SPLINE
SPL {X  -124.075, Y  +778.932, Z    +0.000, E1   -61.393, E3 +26417.862}
SPL {X  -150.653, Y  +735.257, Z    +0.000, E1   -50.160, E3 +26425.541}
SPL {X  -159.377, Y  +706.804, Z    +0.000, E1   -34.828, E3 +26427.184}
SPL {X  -162.134, Y  +688.425, Z    +0.000, E1   -19.100, E3 +26427.121}
SPL {X  -162.803, Y  +675.871, Z    +0.000, E1    -5.469, E3 +26427.305}
SPL {X  -162.820, Y  +671.500, Z    +0.000, E1    +0.000, E3 +26426.873}
SPL {X  -162.820, Y  +669.743, Z    +0.000, E1    +4.352, E3 +26426.669}
SPL {X  -162.820, Y  +665.917, Z    +0.000, E1   +15.272, E3 +26426.663}
SPL {X  -162.820, Y  +661.245, Z    +0.000, E1   +28.879, E3 +26426.504}
SPL {X  -162.820, Y  +654.015, Z    +0.000, E1   +45.814, E3 +26426.651}
SPL {X  -162.820, Y  +641.345, Z    +0.000, E1   +63.138, E3 +26426.698}
SPL {X  -162.820, Y  +620.039, Z    +0.000, E1   +75.979, E3 +26425.308}
SPL {X  -162.820, Y  +571.094, Z    +0.000, E1   +77.089, E3 +26440.487}
SPL {X  -157.487, Y  +339.169, Z    +0.000, E1   +76.425, E3 +26533.591}
SPL {X  -156.386, Y  +335.181, Z    +0.000, E1   +75.555, E3 +26545.652}
SPL {X  -152.710, Y  +324.020, Z    +0.000, E1   +75.365, E3 +26553.462}
SPL {X  -139.497, Y  +296.529, Z    +0.000, E1   +77.231, E3 +26547.034}
ENDSPLINE

SPLINE
SPL {X  -139.792, Y  +297.022, Z    +0.000, E1   +76.273, E3 +26555.729}
ENDSPLINE

SPLINE
SPL {X  -138.933, Y  +295.600, Z    +0.000, E1   +75.173, E3 +26566.212}
SPL {X  -137.186, Y  +292.805, Z    +0.000, E1   +73.993, E3 +26576.802}
SPL {X  -133.270, Y  +286.961, Z    +0.000, E1   +73.739, E3 +26581.515}
SPL {X  -130.283, Y  +282.844, Z    +0.000, E1   +73.297, E3 +26586.407}
SPL {X  -127.795, Y  +279.610, Z    +0.000, E1   +72.860, E3 +26590.537}
SPL {X  -124.650, Y  +275.749, Z    +0.000, E1   +72.674, E3 +26593.456}
SPL {X  -121.687, Y  +272.322, Z    +0.000, E1   +72.100, E3 +26597.765}
SPL {X  -113.980, Y  +264.229, Z    +0.000, E1   +74.120, E3 +26593.903}
SPL {X   -56.216, Y  +227.692, Z    +0.000, E1   +56.267, E3 +26770.627}
ENDSPLINE

SPLINE
SPL {X  -126.995, Y  +278.604, Z    +0.000, E1   +59.937, E3 +26942.868}
SPL {X  -150.196, Y  +317.640, Z    +0.000, E1   +49.956, E3 +26951.323}
SPL {X  -157.261, Y  +338.316, Z    +0.000, E1   +40.017, E3 +26953.018}
SPL {X  -160.924, Y  +355.726, Z    +0.000, E1   +27.715, E3 +26953.459}
SPL {X  -162.423, Y  +369.141, Z    +0.000, E1   +15.207, E3 +26953.894}
SPL {X  -162.811, Y  +378.755, Z    +0.000, E1    +4.616, E3 +26953.808}
SPL {X  -162.820, Y  +382.684, Z    +0.000, E1    -0.227, E3 +26953.363}
SPL {X  -162.820, Y  +387.227, Z    +0.000, E1   -12.320, E3 +26953.118}
SPL {X  -162.820, Y  +392.558, Z    +0.000, E1   -27.778, E3 +26953.154}
SPL {X  -162.820, Y  +400.474, Z    +0.000, E1   -46.251, E3 +26953.018}
SPL {X  -162.820, Y  +414.510, Z    +0.000, E1   -65.115, E3 +26952.461}
SPL {X  -162.820, Y  +465.064, Z    +0.000, E1   -76.269, E3 +26962.309}
SPL {X  -157.184, Y  +715.968, Z    +0.000, E1   -76.600, E3 +27058.266}
SPL {X  -156.461, Y  +718.560, Z    +0.000, E1   -75.553, E3 +27071.686}
SPL {X  -151.911, Y  +732.096, Z    +0.000, E1   -75.235, E3 +27082.240}
SPL {X  -146.569, Y  +744.407, Z    +0.000, E1   -74.677, E3 +27094.044}
SPL {X  -142.375, Y  +752.491, Z    +0.000, E1   -74.335, E3 +27101.072}
SPL {X  -139.539, Y  +757.399, Z    +0.000, E1   -73.892, E3 +27107.269}
SPL {X  -136.017, Y  +762.997, Z    +0.000, E1   -73.579, E3 +27112.452}
SPL {X  -133.089, Y  +767.296, Z    +0.000, E1   -73.251, E3 +27116.910}
SPL {X  -129.985, Y  +771.553, Z    +0.000, E1   -72.801, E3 +27121.904}
SPL {X  -126.581, Y  +775.909, Z    +0.000, E1   -72.426, E3 +27126.215}
SPL {X  -123.329, Y  +779.803, Z    +0.000, E1   -71.936, E3 +27130.597}
SPL {X  -119.291, Y  +784.315, Z    +0.000, E1   -72.148, E3 +27132.009}
SPL {X   -57.587, Y  +825.796, Z    +0.000, E1   -56.753, E3 +27285.771}
ENDSPLINE

SPLINE
SPL {X  -124.075, Y  +778.932, Z    +0.000, E1   -61.393, E3 +27479.400}
SPL {X  -150.653, Y  +735.257, Z    +0.000, E1   -50.160, E3 +27487.079}
SPL {X  -159.377, Y  +706.804, Z    +0.000, E1   -34.828, E3 +27488.723}
SPL {X  -162.134, Y  +688.425, Z    +0.000, E1   -19.100, E3 +27488.659}
SPL {X  -162.803, Y  +675.871, Z    +0.000, E1    -5.469, E3 +27488.843}
SPL {X  -162.820, Y  +671.500, Z    +0.000, E1    +0.000, E3 +27488.411}
SPL {X  -162.820, Y  +669.743, Z    +0.000, E1    +4.352, E3 +27488.207}
SPL {X  -162.820, Y  +665.917, Z    +0.000, E1   +15.272, E3 +27488.202}
SPL {X  -162.820, Y  +661.245, Z    +0.000, E1   +28.879, E3 +27488.043}
SPL {X  -162.820, Y  +654.015, Z    +0.000, E1   +45.814, E3 +27488.190}
SPL {X  -162.820, Y  +641.345, Z    +0.000, E1   +63.138, E3 +27488.237}
SPL {X  -162.820, Y  +620.039, Z    +0.000, E1   +75.979, E3 +27486.847}
SPL {X  -162.820, Y  +571.094, Z    +0.000, E1   +77.089, E3 +27502.025}
SPL {X  -157.487, Y  +339.169, Z    +0.000, E1   +76.425, E3 +27595.129}
SPL {X  -156.386, Y  +335.181, Z    +0.000, E1   +75.555, E3 +27607.190}
SPL {X  -152.710, Y  +324.020, Z    +0.000, E1   +75.365, E3 +27615.000}
SPL {X  -139.497, Y  +296.529, Z    +0.000, E1   +77.231, E3 +27608.572}
ENDSPLINE

SPLINE
SPL {X  -139.792, Y  +297.022, Z    +0.000, E1   +76.273, E3 +27617.267}
ENDSPLINE

SPLINE
SPL {X  -138.933, Y  +295.600, Z    +0.000, E1   +75.173, E3 +27627.750}
SPL {X  -137.186, Y  +292.805, Z    +0.000, E1   +73.993, E3 +27638.340}
SPL {X  -133.270, Y  +286.961, Z    +0.000, E1   +73.739, E3 +27643.054}
SPL {X  -130.283, Y  +282.844, Z    +0.000, E1   +73.297, E3 +27647.946}
SPL {X  -127.795, Y  +279.610, Z    +0.000, E1   +72.860, E3 +27652.076}
SPL {X  -124.650, Y  +275.749, Z    +0.000, E1   +72.674, E3 +27654.994}
SPL {X  -121.687, Y  +272.322, Z    +0.000, E1   +72.100, E3 +27659.304}
SPL {X  -113.980, Y  +264.229, Z    +0.000, E1   +74.120, E3 +27655.442}
SPL {X   -56.216, Y  +227.692, Z    +0.000, E1   +56.267, E3 +27832.166}
ENDSPLINE

SPLINE
SPL {X  -126.995, Y  +278.604, Z    +0.000, E1   +59.937, E3 +28004.406}
SPL {X  -150.196, Y  +317.640, Z    +0.000, E1   +49.956, E3 +28012.861}
SPL {X  -157.261, Y  +338.316, Z    +0.000, E1   +40.017, E3 +28014.556}
SPL {X  -160.924, Y  +355.726, Z    +0.000, E1   +27.715, E3 +28014.997}
SPL {X  -162.423, Y  +369.141, Z    +0.000, E1   +15.207, E3 +28015.432}
SPL {X  -162.811, Y  +378.755, Z    +0.000, E1    +4.616, E3 +28015.347}
SPL {X  -162.820, Y  +382.684, Z    +0.000, E1    -0.227, E3 +28014.902}
SPL {X  -162.820, Y  +387.227, Z    +0.000, E1   -12.320, E3 +28014.656}
SPL {X  -162.820, Y  +392.558, Z    +0.000, E1   -27.778, E3 +28014.692}
SPL {X  -162.820, Y  +400.474, Z    +0.000, E1   -46.251, E3 +28014.556}
SPL {X  -162.820, Y  +414.510, Z    +0.000, E1   -65.115, E3 +28013.999}
SPL {X  -162.820, Y  +465.064, Z    +0.000, E1   -76.269, E3 +28023.847}
SPL {X  -157.184, Y  +715.968, Z    +0.000, E1   -76.600, E3 +28119.805}
SPL {X  -156.461, Y  +718.560, Z    +0.000, E1   -75.553, E3 +28133.225}
SPL {X  -151.911, Y  +732.096, Z    +0.000, E1   -75.235, E3 +28143.779}
SPL {X  -146.569, Y  +744.407, Z    +0.000, E1   -74.677, E3 +28155.583}
SPL {X  -142.375, Y  +752.491, Z    +0.000, E1   -74.335, E3 +28162.610}
SPL {X  -139.539, Y  +757.399, Z    +0.000, E1   -73.892, E3 +28168.808}
SPL {X  -136.017, Y  +762.997, Z    +0.000, E1   -73.579, E3 +28173.990}
SPL {X  -133.089, Y  +767.296, Z    +0.000, E1   -73.251, E3 +28178.448}
SPL {X  -129.985, Y  +771.553, Z    +0.000, E1   -72.801, E3 +28183.442}
SPL {X  -126.581, Y  +775.909, Z    +0.000, E1   -72.426, E3 +28187.753}
SPL {X  -123.329, Y  +779.803, Z    +0.000, E1   -71.936, E3 +28192.135}
SPL {X  -119.291, Y  +784.315, Z    +0.000, E1   -72.148, E3 +28193.547}
SPL {X   -57.587, Y  +825.796, Z    +0.000, E1   -56.753, E3 +28347.309}
ENDSPLINE

SPLINE
SPL {X  -124.075, Y  +778.932, Z    +0.000, E1   -61.393, E3 +28540.938}
SPL {X  -150.653, Y  +735.257, Z    +0.000, E1   -50.160, E3 +28548.618}
SPL {X  -159.377, Y  +706.804, Z    +0.000, E1   -34.828, E3 +28550.261}
SPL {X  -162.134, Y  +688.425, Z    +0.000, E1   -19.100, E3 +28550.198}
SPL {X  -162.803, Y  +675.871, Z    +0.000, E1    -5.469, E3 +28550.382}
SPL {X  -162.820, Y  +671.500, Z    +0.000, E1    +0.000, E3 +28549.950}
SPL {X  -162.820, Y  +669.743, Z    +0.000, E1    +4.352, E3 +28549.746}
SPL {X  -162.820, Y  +665.917, Z    +0.000, E1   +15.272, E3 +28549.740}
SPL {X  -162.820, Y  +661.245, Z    +0.000, E1   +28.879, E3 +28549.581}
SPL {X  -162.820, Y  +654.015, Z    +0.000, E1   +45.814, E3 +28549.728}
SPL {X  -162.820, Y  +641.345, Z    +0.000, E1   +63.138, E3 +28549.775}
SPL {X  -162.820, Y  +620.039, Z    +0.000, E1   +75.979, E3 +28548.385}
SPL {X  -162.820, Y  +571.094, Z    +0.000, E1   +77.089, E3 +28563.564}
SPL {X  -157.487, Y  +339.169, Z    +0.000, E1   +76.425, E3 +28656.668}
SPL {X  -156.386, Y  +335.181, Z    +0.000, E1   +75.555, E3 +28668.729}
SPL {X  -152.710, Y  +324.020, Z    +0.000, E1   +75.365, E3 +28676.539}
SPL {X  -139.497, Y  +296.529, Z    +0.000, E1   +77.231, E3 +28670.111}
ENDSPLINE

SPLINE
SPL {X  -139.792, Y  +297.022, Z    +0.000, E1   +76.273, E3 +28678.806}
ENDSPLINE

SPLINE
SPL {X  -138.933, Y  +295.600, Z    +0.000, E1   +75.173, E3 +28689.289}
SPL {X  -137.186, Y  +292.805, Z    +0.000, E1   +73.993, E3 +28699.879}
SPL {X  -133.270, Y  +286.961, Z    +0.000, E1   +73.739, E3 +28704.592}
SPL {X  -130.283, Y  +282.844, Z    +0.000, E1   +73.297, E3 +28709.484}
SPL {X  -127.795, Y  +279.610, Z    +0.000, E1   +72.860, E3 +28713.614}
SPL {X  -124.650, Y  +275.749, Z    +0.000, E1   +72.674, E3 +28716.533}
SPL {X  -121.687, Y  +272.322, Z    +0.000, E1   +72.100, E3 +28720.842}
SPL {X  -113.980, Y  +264.229, Z    +0.000, E1   +74.120, E3 +28716.980}
SPL {X   -56.216, Y  +227.692, Z    +0.000, E1   +56.267, E3 +28893.704}
ENDSPLINE

SPLINE
SPL {X  -126.995, Y  +278.604, Z    +0.000, E1   +59.937, E3 +29065.945}
SPL {X  -150.196, Y  +317.640, Z    +0.000, E1   +49.956, E3 +29074.400}
SPL {X  -157.261, Y  +338.316, Z    +0.000, E1   +40.017, E3 +29076.095}
SPL {X  -160.924, Y  +355.726, Z    +0.000, E1   +27.715, E3 +29076.535}
SPL {X  -162.423, Y  +369.141, Z    +0.000, E1   +15.207, E3 +29076.971}
SPL {X  -162.811, Y  +378.755, Z    +0.000, E1    +4.616, E3 +29076.885}
SPL {X  -162.820, Y  +382.684, Z    +0.000, E1    -0.227, E3 +29076.440}
SPL {X  -162.820, Y  +387.227, Z    +0.000, E1   -12.320, E3 +29076.195}
SPL {X  -162.820, Y  +392.558, Z    +0.000, E1   -27.778, E3 +29076.231}
SPL {X  -162.820, Y  +400.474, Z    +0.000, E1   -46.251, E3 +29076.095}
SPL {X  -162.820, Y  +414.510, Z    +0.000, E1   -65.115, E3 +29075.538}
SPL {X  -162.820, Y  +465.064, Z    +0.000, E1   -76.269, E3 +29085.386}
SPL {X  -157.184, Y  +715.968, Z    +0.000, E1   -76.600, E3 +29181.343}
SPL {X  -156.461, Y  +718.560, Z    +0.000, E1   -75.553, E3 +29194.763}
SPL {X  -151.911, Y  +732.096, Z    +0.000, E1   -75.235, E3 +29205.317}
SPL {X  -146.569, Y  +744.407, Z    +0.000, E1   -74.677, E3 +29217.121}
SPL {X  -142.375, Y  +752.491, Z    +0.000, E1   -74.335, E3 +29224.149}
SPL {X  -139.539, Y  +757.399, Z    +0.000, E1   -73.892, E3 +29230.346}
SPL {X  -136.017, Y  +762.997, Z    +0.000, E1   -73.579, E3 +29235.529}
SPL {X  -133.089, Y  +767.296, Z    +0.000, E1   -73.251, E3 +29239.987}
SPL {X  -129.985, Y  +771.553, Z    +0.000, E1   -72.801, E3 +29244.981}
SPL {X  -126.581, Y  +775.909, Z    +0.000, E1   -72.426, E3 +29249.292}
SPL {X  -123.329, Y  +779.803, Z    +0.000, E1   -71.936, E3 +29253.674}
SPL {X  -119.291, Y  +784.315, Z    +0.000, E1   -72.148, E3 +29255.085}
SPL {X   -57.587, Y  +825.796, Z    +0.000, E1   -56.753, E3 +29408.848}
ENDSPLINE

SPLINE
SPL {X  -124.075, Y  +778.932, Z    +0.000, E1   -61.393, E3 +29602.477}
SPL {X  -150.653, Y  +735.257, Z    +0.000, E1   -50.160, E3 +29610.156}
SPL {X  -159.377, Y  +706.804, Z    +0.000, E1   -34.828, E3 +29611.800}
SPL {X  -162.134, Y  +688.425, Z    +0.000, E1   -19.100, E3 +29611.736}
SPL {X  -162.803, Y  +675.871, Z    +0.000, E1    -5.469, E3 +29611.920}
SPL {X  -162.820, Y  +671.500, Z    +0.000, E1    +0.000, E3 +29611.488}
SPL {X  -162.820, Y  +669.743, Z    +0.000, E1    +4.352, E3 +29611.284}
SPL {X  -162.820, Y  +665.917, Z    +0.000, E1   +15.272, E3 +29611.279}
SPL {X  -162.820, Y  +661.245, Z    +0.000, E1   +28.879, E3 +29611.120}
SPL {X  -162.820, Y  +654.015, Z    +0.000, E1   +45.814, E3 +29611.267}
SPL {X  -162.820, Y  +641.345, Z    +0.000, E1   +63.138, E3 +29611.314}
SPL {X  -162.820, Y  +620.039, Z    +0.000, E1   +75.979, E3 +29609.924}
SPL {X  -162.820, Y  +571.094, Z    +0.000, E1   +77.089, E3 +29625.102}
SPL {X  -158.110, Y  +341.619, Z    +0.000, E1   +77.339, E3 +29706.752}
SPL {X  -156.597, Y  +335.917, Z    +0.000, E1   +75.680, E3 +29728.595}
SPL {X  -152.710, Y  +324.020, Z    +0.000, E1   +75.365, E3 +29738.077}
SPL {X  -139.497, Y  +296.529, Z    +0.000, E1   +77.231, E3 +29731.649}
ENDSPLINE

SPLINE
SPL {X  -139.792, Y  +297.022, Z    +0.000, E1   +76.273, E3 +29740.344}
ENDSPLINE

SPLINE
SPL {X  -138.933, Y  +295.600, Z    +0.000, E1   +75.173, E3 +29750.827}
SPL {X  -137.186, Y  +292.805, Z    +0.000, E1   +73.993, E3 +29761.417}
SPL {X  -133.270, Y  +286.961, Z    +0.000, E1   +73.739, E3 +29766.131}
SPL {X  -130.283, Y  +282.844, Z    +0.000, E1   +73.297, E3 +29771.023}
SPL {X  -127.795, Y  +279.610, Z    +0.000, E1   +72.860, E3 +29775.153}
SPL {X  -124.650, Y  +275.749, Z    +0.000, E1   +72.674, E3 +29778.071}
SPL {X  -121.687, Y  +272.322, Z    +0.000, E1   +72.100, E3 +29782.381}
SPL {X  -113.980, Y  +264.229, Z    +0.000, E1   +74.120, E3 +29778.519}
SPL {X   -56.216, Y  +227.692, Z    +0.000, E1   +56.267, E3 +29955.243}
ENDSPLINE

SPLINE
SPL {X  -126.995, Y  +278.604, Z    +0.000, E1   +59.937, E3 +30127.483}
SPL {X  -150.196, Y  +317.640, Z    +0.000, E1   +49.956, E3 +30135.938}
SPL {X  -157.261, Y  +338.316, Z    +0.000, E1   +40.017, E3 +30137.633}
SPL {X  -160.924, Y  +355.726, Z    +0.000, E1   +27.715, E3 +30138.074}
SPL {X  -162.423, Y  +369.141, Z    +0.000, E1   +15.207, E3 +30138.509}
SPL {X  -162.811, Y  +378.755, Z    +0.000, E1    +4.616, E3 +30138.424}
SPL {X  -162.820, Y  +382.684, Z    +0.000, E1    -0.227, E3 +30137.978}
SPL {X  -162.820, Y  +385.721, Z    +0.000, E1    -8.371, E3 +30137.794}
SPL {X  -162.820, Y  +388.532, Z    +0.000, E1   -16.412, E3 +30137.681}
SPL {X  -162.820, Y  +392.558, Z    +0.000, E1   -27.778, E3 +30137.769}
SPL {X  -162.820, Y  +400.474, Z    +0.000, E1   -46.251, E3 +30137.633}
SPL {X  -162.820, Y  +414.510, Z    +0.000, E1   -65.115, E3 +30137.076}
SPL {X  -162.820, Y  +465.064, Z    +0.000, E1   -76.269, E3 +30146.924}
SPL {X  -158.097, Y  +712.432, Z    +0.000, E1   -77.677, E3 +30229.312}
SPL {X  -156.557, Y  +718.224, Z    +0.000, E1   -75.715, E3 +30254.448}
SPL {X  -153.015, Y  +729.150, Z    +0.000, E1   -75.312, E3 +30264.391}
SPL {X  -149.053, Y  +739.025, Z    +0.000, E1   -74.952, E3 +30273.186}
SPL {X  -145.525, Y  +746.527, Z    +0.000, E1   -74.526, E3 +30280.980}
SPL {X  -142.375, Y  +752.491, Z    +0.000, E1   -74.335, E3 +30285.687}
SPL {X  -139.539, Y  +757.399, Z    +0.000, E1   -73.892, E3 +30291.885}
SPL {X  -136.017, Y  +762.997, Z    +0.000, E1   -73.579, E3 +30297.067}
SPL {X  -133.089, Y  +767.296, Z    +0.000, E1   -73.251, E3 +30301.525}
SPL {X  -129.985, Y  +771.553, Z    +0.000, E1   -72.801, E3 +30306.519}
SPL {X  -126.581, Y  +775.909, Z    +0.000, E1   -72.426, E3 +30310.830}
SPL {X  -123.329, Y  +779.803, Z    +0.000, E1   -71.936, E3 +30315.212}
SPL {X  -119.291, Y  +784.315, Z    +0.000, E1   -72.148, E3 +30316.624}
SPL {X   -57.587, Y  +825.796, Z    +0.000, E1   -56.753, E3 +30470.386}
ENDSPLINE

SPLINE
SPL {X  -124.075, Y  +778.932, Z    +0.000, E1   -61.393, E3 +30664.015}
SPL {X  -150.653, Y  +735.257, Z    +0.000, E1   -50.160, E3 +30671.695}
SPL {X  -159.377, Y  +706.804, Z    +0.000, E1   -34.828, E3 +30673.338}
SPL {X  -162.134, Y  +688.425, Z    +0.000, E1   -19.100, E3 +30673.275}
SPL {X  -162.803, Y  +675.871, Z    +0.000, E1    -5.469, E3 +30673.459}
SPL {X  -162.820, Y  +671.500, Z    +0.000, E1    +0.000, E3 +30673.027}
SPL {X  -162.820, Y  +669.743, Z    +0.000, E1    +4.352, E3 +30672.822}
SPL {X  -162.820, Y  +665.917, Z    +0.000, E1   +15.272, E3 +30672.817}
SPL {X  -162.820, Y  +659.880, Z    +0.000, E1   +32.256, E3 +30672.728}
SPL {X  -162.820, Y  +652.069, Z    +0.000, E1   +49.663, E3 +30672.754}
SPL {X  -162.820, Y  +641.345, Z    +0.000, E1   +63.138, E3 +30672.852}
SPL {X  -162.820, Y  +620.039, Z    +0.000, E1   +75.979, E3 +30671.462}
SPL {X  -162.820, Y  +571.094, Z    +0.000, E1   +77.089, E3 +30686.641}
SPL {X  -157.487, Y  +339.169, Z    +0.000, E1   +76.425, E3 +30779.745}
SPL {X  -156.386, Y  +335.181, Z    +0.000, E1   +75.555, E3 +30791.805}
SPL {X  -152.710, Y  +324.020, Z    +0.000, E1   +75.365, E3 +30799.616}
SPL {X  -139.497, Y  +296.529, Z    +0.000, E1   +77.231, E3 +30793.188}
ENDSPLINE

SPLINE
SPL {X  -139.792, Y  +297.022, Z    +0.000, E1   +76.273, E3 +30801.883}
ENDSPLINE

SPLINE
SPL {X  -138.933, Y  +295.600, Z    +0.000, E1   +75.173, E3 +30812.365}
SPL {X  -137.186, Y  +292.805, Z    +0.000, E1   +73.993, E3 +30822.956}
SPL {X  -133.270, Y  +286.961, Z    +0.000, E1   +73.739, E3 +30827.669}
SPL {X  -129.057, Y  +281.230, Z    +0.000, E1   +73.118, E3 +30834.577}
SPL {X  -123.859, Y  +274.815, Z    +0.000, E1   +72.511, E3 +30840.962}
SPL {X  -121.018, Y  +271.573, Z    +0.000, E1   +72.049, E3 +30844.479}
SPL {X  -113.980, Y  +264.229, Z    +0.000, E1   +74.120, E3 +30840.057}
SPL {X   -56.216, Y  +227.692, Z    +0.000, E1   +56.267, E3 +31016.781}
ENDSPLINE

SPLINE
SPL {X  -126.995, Y  +278.604, Z    +0.000, E1   +59.937, E3 +31189.021}
SPL {X  -150.196, Y  +317.640, Z    +0.000, E1   +49.956, E3 +31197.477}
SPL {X  -157.261, Y  +338.316, Z    +0.000, E1   +40.017, E3 +31199.172}
SPL {X  -160.924, Y  +355.726, Z    +0.000, E1   +27.715, E3 +31199.612}
SPL {X  -162.423, Y  +369.141, Z    +0.000, E1   +15.207, E3 +31200.048}
SPL {X  -162.811, Y  +378.755, Z    +0.000, E1    +4.616, E3 +31199.962}
SPL {X  -162.820, Y  +382.684, Z    +0.000, E1    -0.227, E3 +31199.517}
SPL {X  -162.820, Y  +385.721, Z    +0.000, E1    -8.371, E3 +31199.332}
SPL {X  -162.820, Y  +388.532, Z    +0.000, E1   -16.412, E3 +31199.219}
SPL {X  -162.820, Y  +392.558, Z    +0.000, E1   -27.778, E3 +31199.308}
SPL {X  -162.820, Y  +398.468, Z    +0.000, E1   -42.446, E3 +31199.158}
SPL {X  -162.820, Y  +404.415, Z    +0.000, E1   -53.236, E3 +31199.198}
SPL {X  -162.820, Y  +414.510, Z    +0.000, E1   -65.115, E3 +31198.615}
SPL {X  -162.820, Y  +457.766, Z    +0.000, E1   -75.929, E3 +31206.451}
SPL {X  -162.820, Y  +471.144, Z    +0.000, E1   -76.496, E3 +31210.140}
SPL {X  -158.097, Y  +712.432, Z    +0.000, E1   -77.677, E3 +31290.850}
SPL {X  -156.557, Y  +718.224, Z    +0.000, E1   -75.715, E3 +31315.987}
SPL {X  -153.015, Y  +729.150, Z    +0.000, E1   -75.312, E3 +31325.929}
SPL {X  -149.053, Y  +739.025, Z    +0.000, E1   -74.952, E3 +31334.725}
SPL {X  -144.053, Y  +749.389, Z    +0.000, E1   -74.457, E3 +31344.716}
SPL {X  -139.539, Y  +757.399, Z    +0.000, E1   -73.892, E3 +31353.423}
SPL {X  -136.017, Y  +762.997, Z    +0.000, E1   -73.579, E3 +31358.606}
SPL {X  -133.089, Y  +767.296, Z    +0.000, E1   -73.251, E3 +31363.064}
SPL {X  -129.985, Y  +771.553, Z    +0.000, E1   -72.801, E3 +31368.057}
SPL {X  -126.581, Y  +775.909, Z    +0.000, E1   -72.426, E3 +31372.369}
SPL {X  -123.329, Y  +779.803, Z    +0.000, E1   -71.936, E3 +31376.750}
SPL {X  -119.291, Y  +784.315, Z    +0.000, E1   -72.148, E3 +31378.162}
SPL {X   -57.587, Y  +825.796, Z    +0.000, E1   -56.753, E3 +31531.925}
ENDSPLINE

SPLINE
SPL {X  -124.075, Y  +778.932, Z    +0.000, E1   -61.393, E3 +31725.554}
SPL {X  -150.653, Y  +735.257, Z    +0.000, E1   -50.160, E3 +31733.233}
SPL {X  -159.377, Y  +706.804, Z    +0.000, E1   -34.828, E3 +31734.876}
SPL {X  -162.134, Y  +688.425, Z    +0.000, E1   -19.100, E3 +31734.813}
SPL {X  -162.803, Y  +675.871, Z    +0.000, E1    -5.469, E3 +31734.997}
SPL {X  -162.820, Y  +671.500, Z    +0.000, E1    +0.000, E3 +31734.565}
SPL {X  -162.820, Y  +669.743, Z    +0.000, E1    +4.352, E3 +31734.361}
SPL {X  -162.820, Y  +665.917, Z    +0.000, E1   +15.272, E3 +31734.355}
SPL {X  -162.820, Y  +661.245, Z    +0.000, E1   +28.879, E3 +31734.197}
SPL {X  -162.820, Y  +654.015, Z    +0.000, E1   +45.814, E3 +31734.344}
SPL {X  -162.820, Y  +641.345, Z    +0.000, E1   +63.138, E3 +31734.391}
SPL {X  -162.820, Y  +620.039, Z    +0.000, E1   +75.979, E3 +31733.001}
SPL {X  -162.820, Y  +571.094, Z    +0.000, E1   +77.089, E3 +31748.179}
SPL {X  -157.487, Y  +339.169, Z    +0.000, E1   +76.425, E3 +31841.283}
SPL {X  -156.386, Y  +335.181, Z    +0.000, E1   +75.555, E3 +31853.344}
SPL {X  -152.710, Y  +324.020, Z    +0.000, E1   +75.365, E3 +31861.154}
SPL {X  -139.497, Y  +296.529, Z    +0.000, E1   +77.231, E3 +31854.726}
ENDSPLINE

SPLINE
SPL {X  -139.792, Y  +297.022, Z    +0.000, E1   +76.273, E3 +31863.421}
ENDSPLINE

SPLINE
SPL {X  -138.933, Y  +295.600, Z    +0.000, E1   +75.173, E3 +31873.904}
SPL {X  -137.186, Y  +292.805, Z    +0.000, E1   +73.993, E3 +31884.494}
SPL {X  -133.270, Y  +286.961, Z    +0.000, E1   +73.739, E3 +31889.208}
SPL {X  -130.283, Y  +282.844, Z    +0.000, E1   +73.297, E3 +31894.100}
SPL {X  -127.795, Y  +279.610, Z    +0.000, E1   +72.860, E3 +31898.230}
SPL {X  -124.650, Y  +275.749, Z    +0.000, E1   +72.674, E3 +31901.148}
SPL {X  -121.687, Y  +272.322, Z    +0.000, E1   +72.100, E3 +31905.457}
SPL {X  -113.980, Y  +264.229, Z    +0.000, E1   +74.120, E3 +31901.596}
SPL {X   -56.216, Y  +227.692, Z    +0.000, E1   +56.267, E3 +32078.320}
ENDSPLINE

SPLINE
SPL {X  -126.995, Y  +278.604, Z    +0.000, E1   +59.937, E3 +32250.560}
SPL {X  -150.196, Y  +317.640, Z    +0.000, E1   +49.956, E3 +32259.015}
SPL {X  -157.261, Y  +338.316, Z    +0.000, E1   +40.017, E3 +32260.710}
SPL {X  -160.924, Y  +355.726, Z    +0.000, E1   +27.715, E3 +32261.151}
SPL {X  -162.423, Y  +369.141, Z    +0.000, E1   +15.207, E3 +32261.586}
SPL {X  -162.811, Y  +378.755, Z    +0.000, E1    +4.616, E3 +32261.501}
SPL {X  -162.820, Y  +382.684, Z    +0.000, E1    -0.227, E3 +32261.055}
SPL {X  -162.820, Y  +385.721, Z    +0.000, E1    -8.371, E3 +32260.871}
SPL {X  -162.820, Y  +388.532, Z    +0.000, E1   -16.412, E3 +32260.757}
SPL {X  -162.820, Y  +392.558, Z    +0.000, E1   -27.778, E3 +32260.846}
SPL {X  -162.820, Y  +400.474, Z    +0.000, E1   -46.251, E3 +32260.710}
SPL {X  -162.820, Y  +414.510, Z    +0.000, E1   -65.115, E3 +32260.153}
SPL {X  -162.820, Y  +465.064, Z    +0.000, E1   -76.269, E3 +32270.001}
SPL {X  -158.097, Y  +712.432, Z    +0.000, E1   -77.677, E3 +32352.389}
SPL {X  -156.557, Y  +718.224, Z    +0.000, E1   -75.715, E3 +32377.525}
SPL {X  -153.015, Y  +729.150, Z    +0.000, E1   -75.312, E3 +32387.468}
SPL {X  -149.053, Y  +739.025, Z    +0.000, E1   -74.952, E3 +32396.263}
SPL {X  -145.525, Y  +746.527, Z    +0.000, E1   -74.526, E3 +32404.057}
SPL {X  -142.375, Y  +752.491, Z    +0.000, E1   -74.335, E3 +32408.764}
SPL {X  -139.539, Y  +757.399, Z    +0.000, E1   -73.892, E3 +32414.962}
SPL {X  -136.017, Y  +762.997, Z    +0.000, E1   -73.579, E3 +32420.144}
SPL {X  -133.089, Y  +767.296, Z    +0.000, E1   -73.251, E3 +32424.602}
SPL {X  -129.985, Y  +771.553, Z    +0.000, E1   -72.801, E3 +32429.596}
SPL {X  -126.581, Y  +775.909, Z    +0.000, E1   -72.426, E3 +32433.907}
SPL {X  -123.329, Y  +779.803, Z    +0.000, E1   -71.936, E3 +32438.289}
SPL {X  -119.291, Y  +784.315, Z    +0.000, E1   -72.148, E3 +32439.701}
SPL {X   -57.587, Y  +825.796, Z    +0.000, E1   -56.753, E3 +32593.463}
ENDSPLINE

SPLINE
SPL {X  -124.075, Y  +778.932, Z    +0.000, E1   -61.393, E3 +32787.092}
SPL {X  -147.028, Y  +743.450, Z    +0.000, E1   -53.078, E3 +32793.829}
SPL {X  -152.552, Y  +730.406, Z    +0.000, E1   -48.136, E3 +32795.247}
SPL {X  -159.377, Y  +706.804, Z    +0.000, E1   -34.828, E3 +32796.415}
SPL {X  -162.134, Y  +688.425, Z    +0.000, E1   -19.100, E3 +32796.352}
SPL {X  -162.803, Y  +675.871, Z    +0.000, E1    -5.469, E3 +32796.536}
SPL {X  -162.820, Y  +671.500, Z    +0.000, E1    +0.000, E3 +32796.104}
SPL {X  -162.820, Y  +669.743, Z    +0.000, E1    +4.352, E3 +32795.899}
SPL {X  -162.820, Y  +665.917, Z    +0.000, E1   +15.272, E3 +32795.894}
SPL {X  -162.820, Y  +661.245, Z    +0.000, E1   +28.879, E3 +32795.735}
SPL {X  -162.820, Y  +654.015, Z    +0.000, E1   +45.814, E3 +32795.882}
SPL {X  -162.820, Y  +641.345, Z    +0.000, E1   +63.138, E3 +32795.929}
SPL {X  -162.820, Y  +620.039, Z    +0.000, E1   +75.979, E3 +32794.539}
SPL {X  -162.820, Y  +571.094, Z    +0.000, E1   +77.089, E3 +32809.718}
SPL {X  -157.487, Y  +339.169, Z    +0.000, E1   +76.425, E3 +32902.822}
SPL {X  -156.386, Y  +335.181, Z    +0.000, E1   +75.555, E3 +32914.882}
SPL {X  -152.710, Y  +324.020, Z    +0.000, E1   +75.365, E3 +32922.693}
SPL {X  -139.497, Y  +296.529, Z    +0.000, E1   +77.231, E3 +32916.264}
ENDSPLINE

SPLINE
SPL {X  -139.520, Y  +296.568, Z    +0.000, E1   +75.884, E3 +32928.912}
ENDSPLINE

SPLINE
SPL {X  -138.554, Y  +294.984, Z    +0.000, E1   +74.772, E3 +32938.793}
SPL {X  -137.186, Y  +292.805, Z    +0.000, E1   +73.993, E3 +32946.033}
SPL {X  -133.270, Y  +286.961, Z    +0.000, E1   +73.739, E3 +32950.746}
SPL {X  -130.283, Y  +282.844, Z    +0.000, E1   +73.297, E3 +32955.638}
SPL {X  -127.795, Y  +279.610, Z    +0.000, E1   +72.860, E3 +32959.768}
SPL {X  -124.650, Y  +275.749, Z    +0.000, E1   +72.674, E3 +32962.687}
SPL {X  -121.687, Y  +272.322, Z    +0.000, E1   +72.100, E3 +32966.996}
SPL {X  -113.980, Y  +264.229, Z    +0.000, E1   +74.120, E3 +32963.134}
SPL {X   -56.216, Y  +227.692, Z    +0.000, E1   +56.267, E3 +33139.858}
ENDSPLINE

SPLINE
SPL {X  -126.995, Y  +278.604, Z    +0.000, E1   +59.937, E3 +33312.098}
SPL {X  -150.196, Y  +317.640, Z    +0.000, E1   +49.956, E3 +33320.553}
SPL {X  -157.261, Y  +338.316, Z    +0.000, E1   +40.017, E3 +33322.249}
SPL {X  -160.924, Y  +355.726, Z    +0.000, E1   +27.715, E3 +33322.689}
SPL {X  -162.423, Y  +369.141, Z    +0.000, E1   +15.207, E3 +33323.125}
SPL {X  -162.811, Y  +378.755, Z    +0.000, E1    +4.616, E3 +33323.039}
SPL {X  -162.820, Y  +382.684, Z    +0.000, E1    -0.227, E3 +33322.594}
SPL {X  -162.820, Y  +387.227, Z    +0.000, E1   -12.320, E3 +33322.349}
SPL {X  -162.820, Y  +392.558, Z    +0.000, E1   -27.778, E3 +33322.385}
SPL {X  -162.820, Y  +400.474, Z    +0.000, E1   -46.251, E3 +33322.248}
SPL {X  -162.820, Y  +414.510, Z    +0.000, E1   -65.115, E3 +33321.692}
SPL {X  -162.820, Y  +465.064, Z    +0.000, E1   -76.269, E3 +33331.540}
SPL {X  -157.184, Y  +715.968, Z    +0.000, E1   -76.600, E3 +33427.497}
SPL {X  -156.461, Y  +718.560, Z    +0.000, E1   -75.553, E3 +33440.917}
SPL {X  -151.911, Y  +732.096, Z    +0.000, E1   -75.235, E3 +33451.471}
SPL {X  -146.569, Y  +744.407, Z    +0.000, E1   -74.677, E3 +33463.275}
SPL {X  -142.375, Y  +752.491, Z    +0.000, E1   -74.335, E3 +33470.303}
SPL {X  -139.539, Y  +757.399, Z    +0.000, E1   -73.892, E3 +33476.500}
SPL {X  -136.017, Y  +762.997, Z    +0.000, E1   -73.579, E3 +33481.683}
SPL {X  -133.089, Y  +767.296, Z    +0.000, E1   -73.251, E3 +33486.141}
SPL {X  -129.985, Y  +771.553, Z    +0.000, E1   -72.801, E3 +33491.134}
SPL {X  -126.581, Y  +775.909, Z    +0.000, E1   -72.426, E3 +33495.446}
SPL {X  -122.528, Y  +780.725, Z    +0.000, E1   -71.905, E3 +33500.466}
SPL {X  -116.189, Y  +787.563, Z    +0.000, E1   -72.978, E3 +33499.750}
SPL {X   -59.356, Y  +825.116, Z    +0.000, E1   -57.613, E3 +33635.895}
SPL {X   -56.547, Y  +826.185, Z    +0.000, E1   -55.989, E3 +33702.445}
ENDSPLINE

SPLINE
SPL {X  -124.075, Y  +778.932, Z    +0.000, E1   -61.393, E3 +33848.631}
SPL {X  -150.653, Y  +735.257, Z    +0.000, E1   -50.160, E3 +33856.310}
SPL {X  -159.377, Y  +706.804, Z    +0.000, E1   -34.828, E3 +33857.953}
SPL {X  -162.134, Y  +688.425, Z    +0.000, E1   -19.100, E3 +33857.890}
SPL {X  -162.734, Y  +678.779, Z    +0.000, E1    -8.745, E3 +33858.029}
SPL {X  -162.820, Y  +671.589, Z    +0.000, E1    -0.221, E3 +33857.664}
SPL {X  -162.820, Y  +669.743, Z    +0.000, E1    +4.352, E3 +33857.438}
SPL {X  -162.820, Y  +665.917, Z    +0.000, E1   +15.272, E3 +33857.432}
SPL {X  -162.820, Y  +661.245, Z    +0.000, E1   +28.879, E3 +33857.274}
SPL {X  -162.820, Y  +654.015, Z    +0.000, E1   +45.814, E3 +33857.421}
SPL {X  -162.820, Y  +641.345, Z    +0.000, E1   +63.138, E3 +33857.468}
SPL {X  -162.820, Y  +620.039, Z    +0.000, E1   +75.979, E3 +33856.078}
SPL {X  -162.820, Y  +571.094, Z    +0.000, E1   +77.089, E3 +33871.256}
SPL {X  -157.487, Y  +339.169, Z    +0.000, E1   +76.425, E3 +33964.360}
SPL {X  -156.386, Y  +335.181, Z    +0.000, E1   +75.555, E3 +33976.421}
SPL {X  -152.710, Y  +324.020, Z    +0.000, E1   +75.365, E3 +33984.231}
SPL {X  -139.497, Y  +296.529, Z    +0.000, E1   +77.231, E3 +33977.803}
ENDSPLINE

SPLINE
SPL {X  -139.792, Y  +297.022, Z    +0.000, E1   +76.273, E3 +33986.498}
ENDSPLINE

SPLINE
SPL {X  -138.933, Y  +295.600, Z    +0.000, E1   +75.173, E3 +33996.981}
SPL {X  -137.186, Y  +292.805, Z    +0.000, E1   +73.993, E3 +34007.571}
SPL {X  -133.270, Y  +286.961, Z    +0.000, E1   +73.739, E3 +34012.285}
SPL {X  -129.057, Y  +281.230, Z    +0.000, E1   +73.118, E3 +34019.192}
SPL {X  -124.650, Y  +275.749, Z    +0.000, E1   +72.674, E3 +34024.225}
SPL {X  -121.687, Y  +272.322, Z    +0.000, E1   +72.100, E3 +34028.534}
SPL {X  -113.980, Y  +264.229, Z    +0.000, E1   +74.120, E3 +34024.673}
SPL {X   -56.216, Y  +227.692, Z    +0.000, E1   +56.267, E3 +34201.397}
ENDSPLINE

SPLINE
SPL {X  -126.995, Y  +278.604, Z    +0.000, E1   +59.937, E3 +34373.637}
SPL {X  -150.196, Y  +317.640, Z    +0.000, E1   +49.956, E3 +34382.092}
SPL {X  -157.261, Y  +338.316, Z    +0.000, E1   +40.017, E3 +34383.787}
SPL {X  -160.924, Y  +355.726, Z    +0.000, E1   +27.715, E3 +34384.228}
SPL {X  -162.423, Y  +369.141, Z    +0.000, E1   +15.207, E3 +34384.663}
SPL {X  -162.811, Y  +378.755, Z    +0.000, E1    +4.616, E3 +34384.578}
SPL {X  -162.820, Y  +382.684, Z    +0.000, E1    -0.227, E3 +34384.132}
SPL {X  -162.820, Y  +385.721, Z    +0.000, E1    -8.371, E3 +34383.948}
SPL {X  -162.820, Y  +388.532, Z    +0.000, E1   -16.412, E3 +34383.834}
SPL {X  -162.820, Y  +392.558, Z    +0.000, E1   -27.778, E3 +34383.923}
SPL {X  -162.820, Y  +400.474, Z    +0.000, E1   -46.251, E3 +34383.787}
SPL {X  -162.820, Y  +414.510, Z    +0.000, E1   -65.115, E3 +34383.230}
SPL {X  -162.820, Y  +465.064, Z    +0.000, E1   -76.269, E3 +34393.078}
SPL {X  -157.184, Y  +715.968, Z    +0.000, E1   -76.600, E3 +34489.036}
SPL {X  -156.461, Y  +718.560, Z    +0.000, E1   -75.553, E3 +34502.455}
SPL {X  -153.015, Y  +729.150, Z    +0.000, E1   -75.312, E3 +34510.544}
SPL {X  -149.053, Y  +739.025, Z    +0.000, E1   -74.952, E3 +34519.340}
SPL {X  -144.053, Y  +749.389, Z    +0.000, E1   -74.457, E3 +34529.332}
SPL {X  -139.539, Y  +757.399, Z    +0.000, E1   -73.892, E3 +34538.039}
SPL {X  -136.017, Y  +762.997, Z    +0.000, E1   -73.579, E3 +34543.221}
SPL {X  -133.089, Y  +767.296, Z    +0.000, E1   -73.251, E3 +34547.679}
SPL {X  -129.985, Y  +771.553, Z    +0.000, E1   -72.801, E3 +34552.673}
SPL {X  -126.581, Y  +775.909, Z    +0.000, E1   -72.426, E3 +34556.984}
SPL {X  -122.528, Y  +780.725, Z    +0.000, E1   -71.905, E3 +34562.004}
SPL {X  -116.189, Y  +787.563, Z    +0.000, E1   -72.978, E3 +34561.288}
SPL {X   -59.356, Y  +825.116, Z    +0.000, E1   -57.613, E3 +34697.433}
SPL {X   -56.547, Y  +826.185, Z    +0.000, E1   -55.989, E3 +34763.983}
ENDSPLINE

SPLINE
SPL {X  -124.075, Y  +778.932, Z    +0.000, E1   -61.393, E3 +34910.169}
SPL {X  -150.653, Y  +735.257, Z    +0.000, E1   -50.160, E3 +34917.848}
SPL {X  -159.377, Y  +706.804, Z    +0.000, E1   -34.828, E3 +34919.492}
SPL {X  -162.134, Y  +688.425, Z    +0.000, E1   -19.100, E3 +34919.429}
SPL {X  -162.734, Y  +678.779, Z    +0.000, E1    -8.745, E3 +34919.568}
SPL {X  -162.820, Y  +671.589, Z    +0.000, E1    -0.221, E3 +34919.202}
SPL {X  -162.820, Y  +669.743, Z    +0.000, E1    +4.352, E3 +34918.976}
SPL {X  -162.820, Y  +665.917, Z    +0.000, E1   +15.272, E3 +34918.971}
SPL {X  -162.820, Y  +659.880, Z    +0.000, E1   +32.256, E3 +34918.882}
SPL {X  -162.820, Y  +652.069, Z    +0.000, E1   +49.663, E3 +34918.908}
SPL {X  -162.820, Y  +641.345, Z    +0.000, E1   +63.138, E3 +34919.006}
SPL {X  -162.820, Y  +620.039, Z    +0.000, E1   +75.979, E3 +34917.616}
SPL {X  -162.820, Y  +578.479, Z    +0.000, E1   +77.260, E3 +34929.887}
SPL {X  -162.820, Y  +557.052, Z    +0.000, E1   +76.772, E3 +34938.368}
SPL {X  -157.487, Y  +339.169, Z    +0.000, E1   +76.425, E3 +35025.898}
SPL {X  -156.386, Y  +335.181, Z    +0.000, E1   +75.555, E3 +35037.959}
SPL {X  -152.710, Y  +324.020, Z    +0.000, E1   +75.365, E3 +35045.770}
SPL {X  -139.497, Y  +296.529, Z    +0.000, E1   +77.231, E3 +35039.341}
ENDSPLINE

SPLINE
SPL {X  -139.792, Y  +297.022, Z    +0.000, E1   +76.273, E3 +35048.037}
ENDSPLINE

SPLINE
SPL {X  -138.933, Y  +295.600, Z    +0.000, E1   +75.173, E3 +35058.519}
SPL {X  -137.186, Y  +292.805, Z    +0.000, E1   +73.993, E3 +35069.110}
SPL {X  -133.270, Y  +286.961, Z    +0.000, E1   +73.739, E3 +35073.823}
SPL {X  -130.283, Y  +282.844, Z    +0.000, E1   +73.297, E3 +35078.715}
SPL {X  -127.795, Y  +279.610, Z    +0.000, E1   +72.860, E3 +35082.845}
SPL {X  -124.650, Y  +275.749, Z    +0.000, E1   +72.674, E3 +35085.764}
SPL {X  -121.687, Y  +272.322, Z    +0.000, E1   +72.100, E3 +35090.073}
SPL {X  -113.980, Y  +264.229, Z    +0.000, E1   +74.120, E3 +35086.211}
SPL {X   -56.216, Y  +227.692, Z    +0.000, E1   +56.267, E3 +35262.935}
ENDSPLINE

SPLINE
SPL {X  -126.995, Y  +278.604, Z    +0.000, E1   +59.937, E3 +35435.175}
SPL {X  -150.196, Y  +317.640, Z    +0.000, E1   +49.956, E3 +35443.630}
SPL {X  -157.261, Y  +338.316, Z    +0.000, E1   +40.017, E3 +35445.326}
SPL {X  -160.924, Y  +355.726, Z    +0.000, E1   +27.715, E3 +35445.766}
SPL {X  -162.423, Y  +369.141, Z    +0.000, E1   +15.207, E3 +35446.202}
SPL {X  -162.811, Y  +378.755, Z    +0.000, E1    +4.616, E3 +35446.116}
SPL {X  -162.820, Y  +382.684, Z    +0.000, E1    -0.227, E3 +35445.671}
SPL {X  -162.820, Y  +387.227, Z    +0.000, E1   -12.320, E3 +35445.426}
SPL {X  -162.820, Y  +392.558, Z    +0.000, E1   -27.778, E3 +35445.462}
SPL {X  -162.820, Y  +400.474, Z    +0.000, E1   -46.251, E3 +35445.325}
SPL {X  -162.820, Y  +414.510, Z    +0.000, E1   -65.115, E3 +35444.769}
SPL {X  -162.820, Y  +465.064, Z    +0.000, E1   -76.269, E3 +35454.617}
SPL {X  -157.184, Y  +715.968, Z    +0.000, E1   -76.600, E3 +35550.574}
SPL {X  -156.461, Y  +718.560, Z    +0.000, E1   -75.553, E3 +35563.994}
SPL {X  -153.015, Y  +729.150, Z    +0.000, E1   -75.312, E3 +35572.083}
SPL {X  -149.053, Y  +739.025, Z    +0.000, E1   -74.952, E3 +35580.879}
SPL {X  -144.053, Y  +749.389, Z    +0.000, E1   -74.457, E3 +35590.870}
SPL {X  -139.539, Y  +757.399, Z    +0.000, E1   -73.892, E3 +35599.577}
SPL {X  -136.017, Y  +762.997, Z    +0.000, E1   -73.579, E3 +35604.759}
SPL {X  -133.089, Y  +767.296, Z    +0.000, E1   -73.251, E3 +35609.218}
SPL {X  -129.985, Y  +771.553, Z    +0.000, E1   -72.801, E3 +35614.211}
SPL {X  -126.581, Y  +775.909, Z    +0.000, E1   -72.426, E3 +35618.522}
SPL {X  -122.528, Y  +780.725, Z    +0.000, E1   -71.905, E3 +35623.542}
SPL {X  -116.189, Y  +787.563, Z    +0.000, E1   -72.978, E3 +35622.827}
SPL {X   -59.356, Y  +825.116, Z    +0.000, E1   -57.613, E3 +35758.972}
SPL {X   -56.547, Y  +826.185, Z    +0.000, E1   -55.989, E3 +35825.522}
ENDSPLINE

SPLINE
SPL {X  -124.075, Y  +778.932, Z    +0.000, E1   -61.393, E3 +35971.708}
SPL {X  -150.653, Y  +735.257, Z    +0.000, E1   -50.160, E3 +35979.387}
SPL {X  -159.377, Y  +706.804, Z    +0.000, E1   -34.828, E3 +35981.030}
SPL {X  -162.134, Y  +688.425, Z    +0.000, E1   -19.100, E3 +35980.967}
SPL {X  -162.734, Y  +678.779, Z    +0.000, E1    -8.745, E3 +35981.106}
SPL {X  -162.820, Y  +671.589, Z    +0.000, E1    -0.221, E3 +35980.741}
SPL {X  -162.820, Y  +669.743, Z    +0.000, E1    +4.352, E3 +35980.515}
SPL {X  -162.820, Y  +665.917, Z    +0.000, E1   +15.272, E3 +35980.509}
SPL {X  -162.820, Y  +659.880, Z    +0.000, E1   +32.256, E3 +35980.421}
SPL {X  -162.820, Y  +652.069, Z    +0.000, E1   +49.663, E3 +35980.446}
SPL {X  -162.820, Y  +641.345, Z    +0.000, E1   +63.138, E3 +35980.545}
SPL {X  -162.820, Y  +620.039, Z    +0.000, E1   +75.979, E3 +35979.154}
SPL {X  -162.820, Y  +578.479, Z    +0.000, E1   +77.260, E3 +35991.425}
SPL {X  -162.820, Y  +557.052, Z    +0.000, E1   +76.772, E3 +35999.906}
SPL {X  -157.487, Y  +339.169, Z    +0.000, E1   +76.425, E3 +36087.437}
SPL {X  -156.386, Y  +335.181, Z    +0.000, E1   +75.555, E3 +36099.498}
SPL {X  -152.710, Y  +324.020, Z    +0.000, E1   +75.365, E3 +36107.308}
SPL {X  -139.497, Y  +296.529, Z    +0.000, E1   +77.231, E3 +36100.880}
ENDSPLINE

SPLINE
SPL {X  -139.792, Y  +297.022, Z    +0.000, E1   +76.273, E3 +36109.575}
ENDSPLINE

SPLINE
SPL {X  -138.933, Y  +295.600, Z    +0.000, E1   +75.173, E3 +36120.058}
SPL {X  -137.186, Y  +292.805, Z    +0.000, E1   +73.993, E3 +36130.648}
SPL {X  -133.270, Y  +286.961, Z    +0.000, E1   +73.739, E3 +36135.362}
SPL {X  -130.283, Y  +282.844, Z    +0.000, E1   +73.297, E3 +36140.253}
SPL {X  -126.880, Y  +278.461, Z    +0.000, E1   +72.855, E3 +36145.004}
SPL {X  -124.135, Y  +275.140, Z    +0.000, E1   +72.554, E3 +36148.132}
SPL {X  -121.687, Y  +272.322, Z    +0.000, E1   +72.100, E3 +36151.611}
SPL {X  -113.980, Y  +264.229, Z    +0.000, E1   +74.120, E3 +36147.750}
SPL {X   -56.216, Y  +227.692, Z    +0.000, E1   +56.267, E3 +36324.474}
ENDSPLINE

SPLINE
SPL {X  -126.995, Y  +278.604, Z    +0.000, E1   +59.937, E3 +36496.714}
SPL {X  -150.196, Y  +317.640, Z    +0.000, E1   +49.956, E3 +36505.169}
SPL {X  -157.261, Y  +338.316, Z    +0.000, E1   +40.017, E3 +36506.864}
SPL {X  -160.924, Y  +355.726, Z    +0.000, E1   +27.715, E3 +36507.305}
SPL {X  -162.423, Y  +369.141, Z    +0.000, E1   +15.207, E3 +36507.740}
SPL {X  -162.811, Y  +378.755, Z    +0.000, E1    +4.616, E3 +36507.655}
SPL {X  -162.820, Y  +382.684, Z    +0.000, E1    -0.227, E3 +36507.209}
SPL {X  -162.820, Y  +385.721, Z    +0.000, E1    -8.371, E3 +36507.025}
SPL {X  -162.820, Y  +388.532, Z    +0.000, E1   -16.412, E3 +36506.911}
SPL {X  -162.820, Y  +392.558, Z    +0.000, E1   -27.778, E3 +36507.000}
SPL {X  -162.820, Y  +400.474, Z    +0.000, E1   -46.251, E3 +36506.864}
SPL {X  -162.820, Y  +414.510, Z    +0.000, E1   -65.115, E3 +36506.307}
SPL {X  -162.820, Y  +465.064, Z    +0.000, E1   -76.269, E3 +36516.155}
SPL {X  -157.184, Y  +715.968, Z    +0.000, E1   -76.600, E3 +36612.112}
SPL {X  -156.461, Y  +718.560, Z    +0.000, E1   -75.553, E3 +36625.532}
SPL {X  -153.015, Y  +729.150, Z    +0.000, E1   -75.312, E3 +36633.621}
SPL {X  -149.053, Y  +739.025, Z    +0.000, E1   -74.952, E3 +36642.417}
SPL {X  -144.053, Y  +749.389, Z    +0.000, E1   -74.457, E3 +36652.409}
SPL {X  -139.539, Y  +757.399, Z    +0.000, E1   -73.892, E3 +36661.116}
SPL {X  -136.017, Y  +762.997, Z    +0.000, E1   -73.579, E3 +36666.298}
SPL {X  -133.089, Y  +767.296, Z    +0.000, E1   -73.251, E3 +36670.756}
SPL {X  -129.985, Y  +771.553, Z    +0.000, E1   -72.801, E3 +36675.750}
SPL {X  -126.581, Y  +775.909, Z    +0.000, E1   -72.426, E3 +36680.061}
SPL {X  -123.329, Y  +779.803, Z    +0.000, E1   -71.936, E3 +36684.443}
SPL {X  -119.291, Y  +784.315, Z    +0.000, E1   -72.148, E3 +36685.855}
SPL {X   -57.587, Y  +825.796, Z    +0.000, E1   -56.753, E3 +36839.617}
ENDSPLINE

SPLINE
SPL {X  -124.075, Y  +778.932, Z    +0.000, E1   -61.393, E3 +37033.246}
SPL {X  -150.653, Y  +735.257, Z    +0.000, E1   -50.160, E3 +37040.925}
SPL {X  -159.377, Y  +706.804, Z    +0.000, E1   -34.828, E3 +37042.569}
SPL {X  -162.134, Y  +688.425, Z    +0.000, E1   -19.100, E3 +37042.506}
SPL {X  -162.803, Y  +675.871, Z    +0.000, E1    -5.469, E3 +37042.690}
SPL {X  -162.820, Y  +671.500, Z    +0.000, E1    +0.000, E3 +37042.258}
SPL {X  -162.820, Y  +669.743, Z    +0.000, E1    +4.352, E3 +37042.053}
SPL {X  -162.820, Y  +665.917, Z    +0.000, E1   +15.272, E3 +37042.048}
SPL {X  -162.820, Y  +659.880, Z    +0.000, E1   +32.256, E3 +37041.959}
SPL {X  -162.820, Y  +652.069, Z    +0.000, E1   +49.663, E3 +37041.985}
SPL {X  -162.820, Y  +641.345, Z    +0.000, E1   +63.138, E3 +37042.083}
SPL {X  -162.820, Y  +620.039, Z    +0.000, E1   +75.979, E3 +37040.693}
SPL {X  -162.820, Y  +578.479, Z    +0.000, E1   +77.260, E3 +37052.964}
SPL {X  -162.820, Y  +557.052, Z    +0.000, E1   +76.772, E3 +37061.445}
SPL {X  -157.487, Y  +339.169, Z    +0.000, E1   +76.425, E3 +37148.975}
SPL {X  -156.386, Y  +335.181, Z    +0.000, E1   +75.555, E3 +37161.036}
SPL {X  -152.710, Y  +324.020, Z    +0.000, E1   +75.365, E3 +37168.847}
SPL {X  -139.497, Y  +296.529, Z    +0.000, E1   +77.231, E3 +37162.418}
ENDSPLINE

SPLINE
SPL {X  -139.792, Y  +297.022, Z    +0.000, E1   +76.273, E3 +37171.113}
ENDSPLINE

SPLINE
SPL {X  -138.933, Y  +295.600, Z    +0.000, E1   +75.173, E3 +37181.596}
SPL {X  -137.186, Y  +292.805, Z    +0.000, E1   +73.993, E3 +37192.187}
SPL {X  -133.270, Y  +286.961, Z    +0.000, E1   +73.739, E3 +37196.900}
SPL {X  -130.283, Y  +282.844, Z    +0.000, E1   +73.297, E3 +37201.792}
SPL {X  -126.880, Y  +278.461, Z    +0.000, E1   +72.855, E3 +37206.542}
SPL {X  -123.363, Y  +274.237, Z    +0.000, E1   +72.376, E3 +37211.024}
SPL {X  -121.018, Y  +271.573, Z    +0.000, E1   +72.049, E3 +37213.710}
SPL {X  -113.980, Y  +264.229, Z    +0.000, E1   +74.120, E3 +37209.288}
SPL {X   -56.216, Y  +227.692, Z    +0.000, E1   +56.267, E3 +37386.012}
ENDSPLINE

SPLINE
SPL {X  -126.995, Y  +278.604, Z    +0.000, E1   +59.937, E3 +37558.252}
SPL {X  -150.196, Y  +317.640, Z    +0.000, E1   +49.956, E3 +37566.707}
SPL {X  -157.261, Y  +338.316, Z    +0.000, E1   +40.017, E3 +37568.402}
SPL {X  -160.924, Y  +355.726, Z    +0.000, E1   +27.715, E3 +37568.843}
SPL {X  -162.423, Y  +369.141, Z    +0.000, E1   +15.207, E3 +37569.279}
SPL {X  -162.811, Y  +378.755, Z    +0.000, E1    +4.616, E3 +37569.193}
SPL {X  -162.820, Y  +382.684, Z    +0.000, E1    -0.227, E3 +37568.748}
SPL {X  -162.820, Y  +385.721, Z    +0.000, E1    -8.371, E3 +37568.563}
SPL {X  -162.820, Y  +388.532, Z    +0.000, E1   -16.412, E3 +37568.450}
SPL {X  -162.820, Y  +392.558, Z    +0.000, E1   -27.778, E3 +37568.539}
SPL {X  -162.820, Y  +398.468, Z    +0.000, E1   -42.446, E3 +37568.389}
SPL {X  -162.820, Y  +404.415, Z    +0.000, E1   -53.236, E3 +37568.428}
SPL {X  -162.820, Y  +414.510, Z    +0.000, E1   -65.115, E3 +37567.845}
SPL {X  -162.820, Y  +457.766, Z    +0.000, E1   -75.929, E3 +37575.682}
SPL {X  -162.820, Y  +471.144, Z    +0.000, E1   -76.496, E3 +37579.371}
SPL {X  -158.097, Y  +712.432, Z    +0.000, E1   -77.677, E3 +37660.081}
SPL {X  -156.557, Y  +718.224, Z    +0.000, E1   -75.715, E3 +37685.217}
SPL {X  -153.015, Y  +729.150, Z    +0.000, E1   -75.312, E3 +37695.160}
SPL {X  -149.053, Y  +739.025, Z    +0.000, E1   -74.952, E3 +37703.956}
SPL {X  -145.525, Y  +746.527, Z    +0.000, E1   -74.526, E3 +37711.749}
SPL {X  -142.375, Y  +752.491, Z    +0.000, E1   -74.335, E3 +37716.456}
SPL {X  -139.539, Y  +757.399, Z    +0.000, E1   -73.892, E3 +37722.654}
SPL {X  -136.017, Y  +762.997, Z    +0.000, E1   -73.579, E3 +37727.836}
SPL {X  -133.089, Y  +767.296, Z    +0.000, E1   -73.251, E3 +37732.294}
SPL {X  -129.985, Y  +771.553, Z    +0.000, E1   -72.801, E3 +37737.288}
SPL {X  -126.581, Y  +775.909, Z    +0.000, E1   -72.426, E3 +37741.599}
SPL {X  -123.329, Y  +779.803, Z    +0.000, E1   -71.936, E3 +37745.981}
SPL {X  -119.291, Y  +784.315, Z    +0.000, E1   -72.148, E3 +37747.393}
SPL {X   -57.587, Y  +825.796, Z    +0.000, E1   -56.753, E3 +37901.156}
ENDSPLINE

SPLINE
SPL {X  -124.075, Y  +778.932, Z    +0.000, E1   -61.393, E3 +38094.785}
SPL {X  -150.653, Y  +735.257, Z    +0.000, E1   -50.160, E3 +38102.464}
SPL {X  -159.377, Y  +706.804, Z    +0.000, E1   -34.828, E3 +38104.107}
SPL {X  -162.134, Y  +688.425, Z    +0.000, E1   -19.100, E3 +38104.044}
SPL {X  -162.803, Y  +675.871, Z    +0.000, E1    -5.469, E3 +38104.228}
SPL {X  -162.820, Y  +671.500, Z    +0.000, E1    +0.000, E3 +38103.796}
SPL {X  -162.820, Y  +669.743, Z    +0.000, E1    +4.352, E3 +38103.592}
SPL {X  -162.820, Y  +665.917, Z    +0.000, E1   +15.272, E3 +38103.586}
SPL {X  -162.820, Y  +659.880, Z    +0.000, E1   +32.256, E3 +38103.498}
SPL {X  -162.820, Y  +652.069, Z    +0.000, E1   +49.663, E3 +38103.523}
SPL {X  -162.820, Y  +641.345, Z    +0.000, E1   +63.138, E3 +38103.622}
SPL {X  -162.820, Y  +620.039, Z    +0.000, E1   +75.979, E3 +38102.231}
SPL {X  -162.820, Y  +571.094, Z    +0.000, E1   +77.089, E3 +38117.410}
SPL {X  -157.487, Y  +339.169, Z    +0.000, E1   +76.425, E3 +38210.514}
SPL {X  -156.386, Y  +335.181, Z    +0.000, E1   +75.555, E3 +38222.575}
SPL {X  -152.710, Y  +324.020, Z    +0.000, E1   +75.365, E3 +38230.385}
SPL {X  -139.497, Y  +296.529, Z    +0.000, E1   +77.231, E3 +38223.957}
ENDSPLINE

SPLINE
SPL {X  -139.792, Y  +297.022, Z    +0.000, E1   +76.273, E3 +38232.652}
ENDSPLINE

SPLINE
SPL {X  -138.933, Y  +295.600, Z    +0.000, E1   +75.173, E3 +38243.135}
SPL {X  -137.186, Y  +292.805, Z    +0.000, E1   +73.993, E3 +38253.725}
SPL {X  -133.270, Y  +286.961, Z    +0.000, E1   +73.739, E3 +38258.438}
SPL {X  -129.057, Y  +281.230, Z    +0.000, E1   +73.118, E3 +38265.346}
SPL {X  -123.859, Y  +274.815, Z    +0.000, E1   +72.511, E3 +38271.731}
SPL {X  -121.018, Y  +271.573, Z    +0.000, E1   +72.049, E3 +38275.248}
SPL {X  -113.980, Y  +264.229, Z    +0.000, E1   +74.120, E3 +38270.826}
SPL {X   -56.216, Y  +227.692, Z    +0.000, E1   +56.267, E3 +38447.550}
ENDSPLINE

SPLINE
SPL {X  -126.995, Y  +278.604, Z    +0.000, E1   +59.937, E3 +38619.791}
SPL {X  -150.196, Y  +317.640, Z    +0.000, E1   +49.956, E3 +38628.246}
SPL {X  -157.261, Y  +338.316, Z    +0.000, E1   +40.017, E3 +38629.941}
SPL {X  -160.924, Y  +355.726, Z    +0.000, E1   +27.715, E3 +38630.382}
SPL {X  -162.423, Y  +369.141, Z    +0.000, E1   +15.207, E3 +38630.817}
SPL {X  -162.811, Y  +378.755, Z    +0.000, E1    +4.616, E3 +38630.732}
SPL {X  -162.820, Y  +382.684, Z    +0.000, E1    -0.227, E3 +38630.286}
SPL {X  -162.820, Y  +385.721, Z    +0.000, E1    -8.371, E3 +38630.102}
SPL {X  -162.820, Y  +388.532, Z    +0.000, E1   -16.412, E3 +38629.988}
SPL {X  -162.820, Y  +392.558, Z    +0.000, E1   -27.778, E3 +38630.077}
SPL {X  -162.820, Y  +398.468, Z    +0.000, E1   -42.446, E3 +38629.928}
SPL {X  -162.820, Y  +404.415, Z    +0.000, E1   -53.236, E3 +38629.967}
SPL {X  -162.820, Y  +414.510, Z    +0.000, E1   -65.115, E3 +38629.384}
SPL {X  -162.820, Y  +457.766, Z    +0.000, E1   -75.929, E3 +38637.220}
SPL {X  -162.820, Y  +471.144, Z    +0.000, E1   -76.496, E3 +38640.909}
SPL {X  -158.097, Y  +712.432, Z    +0.000, E1   -77.677, E3 +38721.619}
SPL {X  -156.557, Y  +718.224, Z    +0.000, E1   -75.715, E3 +38746.756}
SPL {X  -153.015, Y  +729.150, Z    +0.000, E1   -75.312, E3 +38756.698}
SPL {X  -149.053, Y  +739.025, Z    +0.000, E1   -74.952, E3 +38765.494}
SPL {X  -144.053, Y  +749.389, Z    +0.000, E1   -74.457, E3 +38775.486}
SPL {X  -139.539, Y  +757.399, Z    +0.000, E1   -73.892, E3 +38784.192}
SPL {X  -136.017, Y  +762.997, Z    +0.000, E1   -73.579, E3 +38789.375}
SPL {X  -133.089, Y  +767.296, Z    +0.000, E1   -73.251, E3 +38793.833}
SPL {X  -129.985, Y  +771.553, Z    +0.000, E1   -72.801, E3 +38798.827}
SPL {X  -126.581, Y  +775.909, Z    +0.000, E1   -72.426, E3 +38803.138}
SPL {X  -123.329, Y  +779.803, Z    +0.000, E1   -71.936, E3 +38807.520}
SPL {X  -119.291, Y  +784.315, Z    +0.000, E1   -72.148, E3 +38808.932}
SPL {X   -57.587, Y  +825.796, Z    +0.000, E1   -56.753, E3 +38962.694}
ENDSPLINE

SPLINE
SPL {X  -124.075, Y  +778.932, Z    +0.000, E1   -61.393, E3 +39156.323}
SPL {X  -150.653, Y  +735.257, Z    +0.000, E1   -50.160, E3 +39164.002}
SPL {X  -159.377, Y  +706.804, Z    +0.000, E1   -34.828, E3 +39165.646}
SPL {X  -162.134, Y  +688.425, Z    +0.000, E1   -19.100, E3 +39165.583}
SPL {X  -162.803, Y  +675.871, Z    +0.000, E1    -5.469, E3 +39165.766}
SPL {X  -162.820, Y  +671.500, Z    +0.000, E1    +0.000, E3 +39165.335}
SPL {X  -162.820, Y  +669.743, Z    +0.000, E1    +4.352, E3 +39165.130}
SPL {X  -162.820, Y  +665.917, Z    +0.000, E1   +15.272, E3 +39165.125}
SPL {X  -162.820, Y  +661.245, Z    +0.000, E1   +28.879, E3 +39164.966}
SPL {X  -162.820, Y  +654.015, Z    +0.000, E1   +45.814, E3 +39165.113}
SPL {X  -162.820, Y  +641.345, Z    +0.000, E1   +63.138, E3 +39165.160}
SPL {X  -162.820, Y  +620.039, Z    +0.000, E1   +75.979, E3 +39163.770}
SPL {X  -162.820, Y  +571.094, Z    +0.000, E1   +77.089, E3 +39178.948}
SPL {X  -157.487, Y  +339.169, Z    +0.000, E1   +76.425, E3 +39272.052}
SPL {X  -156.386, Y  +335.181, Z    +0.000, E1   +75.555, E3 +39284.113}
SPL {X  -152.710, Y  +324.020, Z    +0.000, E1   +75.365, E3 +39291.924}
SPL {X  -139.497, Y  +296.529, Z    +0.000, E1   +77.231, E3 +39285.495}
ENDSPLINE

SPLINE
SPL {X  -139.792, Y  +297.022, Z    +0.000, E1   +76.273, E3 +39294.190}
ENDSPLINE

SPLINE
SPL {X  -138.933, Y  +295.600, Z    +0.000, E1   +75.173, E3 +39304.673}
SPL {X  -137.186, Y  +292.805, Z    +0.000, E1   +73.993, E3 +39315.264}
SPL {X  -133.270, Y  +286.961, Z    +0.000, E1   +73.739, E3 +39319.977}
SPL {X  -130.283, Y  +282.844, Z    +0.000, E1   +73.297, E3 +39324.869}
SPL {X  -127.795, Y  +279.610, Z    +0.000, E1   +72.860, E3 +39328.999}
SPL {X  -124.650, Y  +275.749, Z    +0.000, E1   +72.674, E3 +39331.917}
SPL {X  -121.687, Y  +272.322, Z    +0.000, E1   +72.100, E3 +39336.227}
SPL {X  -113.980, Y  +264.229, Z    +0.000, E1   +74.120, E3 +39332.365}
SPL {X   -56.216, Y  +227.692, Z    +0.000, E1   +56.267, E3 +39509.089}
ENDSPLINE

SPLINE
SPL {X  -126.995, Y  +278.604, Z    +0.000, E1   +59.937, E3 +39681.329}
SPL {X  -150.196, Y  +317.640, Z    +0.000, E1   +49.956, E3 +39689.784}
SPL {X  -157.261, Y  +338.316, Z    +0.000, E1   +40.017, E3 +39691.479}
SPL {X  -160.924, Y  +355.726, Z    +0.000, E1   +27.715, E3 +39691.920}
SPL {X  -162.423, Y  +369.141, Z    +0.000, E1   +15.207, E3 +39692.356}
SPL {X  -162.811, Y  +378.755, Z    +0.000, E1    +4.616, E3 +39692.270}
SPL {X  -162.820, Y  +382.684, Z    +0.000, E1    -0.227, E3 +39691.825}
SPL {X  -162.820, Y  +387.227, Z    +0.000, E1   -12.320, E3 +39691.579}
SPL {X  -162.820, Y  +392.558, Z    +0.000, E1   -27.778, E3 +39691.616}
SPL {X  -162.820, Y  +400.474, Z    +0.000, E1   -46.251, E3 +39691.479}
SPL {X  -162.820, Y  +414.510, Z    +0.000, E1   -65.115, E3 +39690.922}
SPL {X  -162.820, Y  +465.064, Z    +0.000, E1   -76.269, E3 +39700.770}
SPL {X  -158.097, Y  +712.432, Z    +0.000, E1   -77.677, E3 +39783.158}
SPL {X  -156.557, Y  +718.224, Z    +0.000, E1   -75.715, E3 +39808.294}
SPL {X  -151.911, Y  +732.096, Z    +0.000, E1   -75.235, E3 +39820.702}
SPL {X  -146.569, Y  +744.407, Z    +0.000, E1   -74.677, E3 +39832.506}
SPL {X  -142.375, Y  +752.491, Z    +0.000, E1   -74.335, E3 +39839.533}
SPL {X  -139.539, Y  +757.399, Z    +0.000, E1   -73.892, E3 +39845.731}
SPL {X  -136.017, Y  +762.997, Z    +0.000, E1   -73.579, E3 +39850.913}
SPL {X  -133.089, Y  +767.296, Z    +0.000, E1   -73.251, E3 +39855.371}
SPL {X  -129.985, Y  +771.553, Z    +0.000, E1   -72.801, E3 +39860.365}
SPL {X  -126.581, Y  +775.909, Z    +0.000, E1   -72.426, E3 +39864.676}
SPL {X  -123.329, Y  +779.803, Z    +0.000, E1   -71.936, E3 +39869.058}
SPL {X  -119.291, Y  +784.315, Z    +0.000, E1   -72.148, E3 +39870.470}
SPL {X   -57.587, Y  +825.796, Z    +0.000, E1   -56.753, E3 +40024.233}
ENDSPLINE

SPLINE
SPL {X  -124.075, Y  +778.932, Z    +0.000, E1   -61.393, E3 +40217.862}
SPL {X  -150.653, Y  +735.257, Z    +0.000, E1   -50.160, E3 +40225.541}
SPL {X  -159.377, Y  +706.804, Z    +0.000, E1   -34.828, E3 +40227.184}
SPL {X  -162.134, Y  +688.425, Z    +0.000, E1   -19.100, E3 +40227.121}
SPL {X  -162.803, Y  +675.871, Z    +0.000, E1    -5.469, E3 +40227.305}
SPL {X  -162.820, Y  +671.500, Z    +0.000, E1    +0.000, E3 +40226.873}
SPL {X  -162.820, Y  +669.743, Z    +0.000, E1    +4.352, E3 +40226.669}
SPL {X  -162.820, Y  +665.917, Z    +0.000, E1   +15.272, E3 +40226.663}
SPL {X  -162.820, Y  +661.245, Z    +0.000, E1   +28.879, E3 +40226.504}
SPL {X  -162.820, Y  +654.015, Z    +0.000, E1   +45.814, E3 +40226.651}
SPL {X  -162.820, Y  +641.345, Z    +0.000, E1   +63.138, E3 +40226.698}
SPL {X  -162.820, Y  +620.039, Z    +0.000, E1   +75.979, E3 +40225.308}
SPL {X  -162.820, Y  +571.094, Z    +0.000, E1   +77.089, E3 +40240.487}
SPL {X  -157.487, Y  +339.169, Z    +0.000, E1   +76.425, E3 +40333.591}
SPL {X  -156.386, Y  +335.181, Z    +0.000, E1   +75.555, E3 +40345.652}
SPL {X  -152.710, Y  +324.020, Z    +0.000, E1   +75.365, E3 +40353.462}
SPL {X  -139.497, Y  +296.529, Z    +0.000, E1   +77.231, E3 +40347.034}
ENDSPLINE

SPLINE
SPL {X  -139.792, Y  +297.022, Z    +0.000, E1   +76.273, E3 +40355.729}
ENDSPLINE

SPLINE
SPL {X  -138.933, Y  +295.600, Z    +0.000, E1   +75.173, E3 +40366.212}
SPL {X  -137.186, Y  +292.805, Z    +0.000, E1   +73.993, E3 +40376.802}
SPL {X  -133.270, Y  +286.961, Z    +0.000, E1   +73.739, E3 +40381.515}
SPL {X  -130.283, Y  +282.844, Z    +0.000, E1   +73.297, E3 +40386.407}
SPL {X  -127.795, Y  +279.610, Z    +0.000, E1   +72.860, E3 +40390.537}
SPL {X  -124.650, Y  +275.749, Z    +0.000, E1   +72.674, E3 +40393.456}
SPL {X  -121.687, Y  +272.322, Z    +0.000, E1   +72.100, E3 +40397.765}
SPL {X  -113.980, Y  +264.229, Z    +0.000, E1   +74.120, E3 +40393.903}
SPL {X   -56.216, Y  +227.692, Z    +0.000, E1   +56.267, E3 +40570.627}
ENDSPLINE

SPLINE
SPL {X  -126.995, Y  +278.604, Z    +0.000, E1   +59.937, E3 +40742.868}
SPL {X  -150.196, Y  +317.640, Z    +0.000, E1   +49.956, E3 +40751.323}
SPL {X  -157.261, Y  +338.316, Z    +0.000, E1   +40.017, E3 +40753.018}
SPL {X  -160.924, Y  +355.726, Z    +0.000, E1   +27.715, E3 +40753.459}
SPL {X  -162.423, Y  +369.141, Z    +0.000, E1   +15.207, E3 +40753.894}
SPL {X  -162.811, Y  +378.755, Z    +0.000, E1    +4.616, E3 +40753.808}
SPL {X  -162.820, Y  +382.684, Z    +0.000, E1    -0.227, E3 +40753.363}
SPL {X  -162.820, Y  +387.227, Z    +0.000, E1   -12.320, E3 +40753.118}
SPL {X  -162.820, Y  +392.558, Z    +0.000, E1   -27.778, E3 +40753.154}
SPL {X  -162.820, Y  +400.474, Z    +0.000, E1   -46.251, E3 +40753.018}
SPL {X  -162.820, Y  +414.510, Z    +0.000, E1   -65.115, E3 +40752.461}
SPL {X  -162.820, Y  +465.064, Z    +0.000, E1   -76.269, E3 +40762.309}
SPL {X  -157.184, Y  +715.968, Z    +0.000, E1   -76.600, E3 +40858.266}
SPL {X  -156.461, Y  +718.560, Z    +0.000, E1   -75.553, E3 +40871.686}
SPL {X  -151.911, Y  +732.096, Z    +0.000, E1   -75.235, E3 +40882.240}
SPL {X  -146.569, Y  +744.407, Z    +0.000, E1   -74.677, E3 +40894.044}
SPL {X  -142.375, Y  +752.491, Z    +0.000, E1   -74.335, E3 +40901.072}
SPL {X  -139.539, Y  +757.399, Z    +0.000, E1   -73.892, E3 +40907.269}
SPL {X  -136.017, Y  +762.997, Z    +0.000, E1   -73.579, E3 +40912.452}
SPL {X  -133.089, Y  +767.296, Z    +0.000, E1   -73.251, E3 +40916.910}
SPL {X  -129.985, Y  +771.553, Z    +0.000, E1   -72.801, E3 +40921.904}
SPL {X  -126.581, Y  +775.909, Z    +0.000, E1   -72.426, E3 +40926.215}
SPL {X  -123.329, Y  +779.803, Z    +0.000, E1   -71.936, E3 +40930.597}
SPL {X  -119.291, Y  +784.315, Z    +0.000, E1   -72.148, E3 +40932.009}
SPL {X   -57.587, Y  +825.796, Z    +0.000, E1   -56.753, E3 +41085.771}
ENDSPLINE

SPLINE
SPL {X  -124.075, Y  +778.932, Z    +0.000, E1   -61.393, E3 +41279.400}
SPL {X  -150.653, Y  +735.257, Z    +0.000, E1   -50.160, E3 +41287.079}
SPL {X  -159.377, Y  +706.804, Z    +0.000, E1   -34.828, E3 +41288.723}
SPL {X  -162.134, Y  +688.425, Z    +0.000, E1   -19.100, E3 +41288.659}
SPL {X  -162.803, Y  +675.871, Z    +0.000, E1    -5.469, E3 +41288.843}
SPL {X  -162.820, Y  +671.500, Z    +0.000, E1    +0.000, E3 +41288.411}
SPL {X  -162.820, Y  +669.743, Z    +0.000, E1    +4.352, E3 +41288.207}
SPL {X  -162.820, Y  +665.917, Z    +0.000, E1   +15.272, E3 +41288.202}
SPL {X  -162.820, Y  +661.245, Z    +0.000, E1   +28.879, E3 +41288.043}
SPL {X  -162.820, Y  +654.015, Z    +0.000, E1   +45.814, E3 +41288.190}
SPL {X  -162.820, Y  +641.345, Z    +0.000, E1   +63.138, E3 +41288.237}
SPL {X  -162.820, Y  +620.039, Z    +0.000, E1   +75.979, E3 +41286.847}
SPL {X  -162.820, Y  +578.479, Z    +0.000, E1   +77.260, E3 +41299.117}
SPL {X  -162.820, Y  +557.052, Z    +0.000, E1   +76.772, E3 +41307.599}
SPL {X  -157.487, Y  +339.169, Z    +0.000, E1   +76.425, E3 +41395.129}
SPL {X  -156.386, Y  +335.181, Z    +0.000, E1   +75.555, E3 +41407.190}
SPL {X  -152.710, Y  +324.020, Z    +0.000, E1   +75.365, E3 +41415.000}
SPL {X  -139.497, Y  +296.529, Z    +0.000, E1   +77.231, E3 +41408.572}
ENDSPLINE

SPLINE
SPL {X  -139.792, Y  +297.022, Z    +0.000, E1   +76.273, E3 +41417.267}
ENDSPLINE

SPLINE
SPL {X  -138.933, Y  +295.600, Z    +0.000, E1   +75.173, E3 +41427.750}
SPL {X  -137.186, Y  +292.805, Z    +0.000, E1   +73.993, E3 +41438.340}
SPL {X  -133.270, Y  +286.961, Z    +0.000, E1   +73.739, E3 +41443.054}
SPL {X  -130.283, Y  +282.844, Z    +0.000, E1   +73.297, E3 +41447.946}
SPL {X  -127.795, Y  +279.610, Z    +0.000, E1   +72.860, E3 +41452.076}
SPL {X  -124.650, Y  +275.749, Z    +0.000, E1   +72.674, E3 +41454.994}
SPL {X  -121.687, Y  +272.322, Z    +0.000, E1   +72.100, E3 +41459.304}
SPL {X  -113.980, Y  +264.229, Z    +0.000, E1   +74.120, E3 +41455.442}
SPL {X   -56.216, Y  +227.692, Z    +0.000, E1   +56.267, E3 +41632.166}
ENDSPLINE

SPLINE
SPL {X  -126.995, Y  +278.604, Z    +0.000, E1   +59.937, E3 +41804.406}
SPL {X  -150.196, Y  +317.640, Z    +0.000, E1   +49.956, E3 +41812.861}
SPL {X  -157.261, Y  +338.316, Z    +0.000, E1   +40.017, E3 +41814.556}
SPL {X  -160.924, Y  +355.726, Z    +0.000, E1   +27.715, E3 +41814.997}
SPL {X  -162.423, Y  +369.141, Z    +0.000, E1   +15.207, E3 +41815.432}
SPL {X  -162.811, Y  +378.755, Z    +0.000, E1    +4.616, E3 +41815.347}
SPL {X  -162.820, Y  +382.684, Z    +0.000, E1    -0.227, E3 +41814.902}
SPL {X  -162.820, Y  +385.721, Z    +0.000, E1    -8.371, E3 +41814.717}
SPL {X  -162.820, Y  +388.532, Z    +0.000, E1   -16.412, E3 +41814.604}
SPL {X  -162.820, Y  +392.558, Z    +0.000, E1   -27.778, E3 +41814.692}
SPL {X  -162.820, Y  +400.474, Z    +0.000, E1   -46.251, E3 +41814.556}
SPL {X  -162.820, Y  +414.510, Z    +0.000, E1   -65.115, E3 +41813.999}
SPL {X  -162.820, Y  +465.064, Z    +0.000, E1   -76.269, E3 +41823.847}
SPL {X  -158.097, Y  +712.432, Z    +0.000, E1   -77.677, E3 +41906.235}
SPL {X  -156.557, Y  +718.224, Z    +0.000, E1   -75.715, E3 +41931.371}
SPL {X  -153.015, Y  +729.150, Z    +0.000, E1   -75.312, E3 +41941.314}
SPL {X  -149.053, Y  +739.025, Z    +0.000, E1   -74.952, E3 +41950.109}
SPL {X  -145.525, Y  +746.527, Z    +0.000, E1   -74.526, E3 +41957.903}
SPL {X  -142.375, Y  +752.491, Z    +0.000, E1   -74.335, E3 +41962.610}
SPL {X  -139.539, Y  +757.399, Z    +0.000, E1   -73.892, E3 +41968.808}
SPL {X  -136.017, Y  +762.997, Z    +0.000, E1   -73.579, E3 +41973.990}
SPL {X  -133.089, Y  +767.296, Z    +0.000, E1   -73.251, E3 +41978.448}
SPL {X  -129.985, Y  +771.553, Z    +0.000, E1   -72.801, E3 +41983.442}
SPL {X  -126.581, Y  +775.909, Z    +0.000, E1   -72.426, E3 +41987.753}
SPL {X  -123.329, Y  +779.803, Z    +0.000, E1   -71.936, E3 +41992.135}
SPL {X  -119.291, Y  +784.315, Z    +0.000, E1   -72.148, E3 +41993.547}
SPL {X   -57.587, Y  +825.796, Z    +0.000, E1   -56.753, E3 +42147.309}
ENDSPLINE

SPLINE
SPL {X  -124.075, Y  +778.932, Z    +0.000, E1   -61.393, E3 +42340.938}
SPL {X  -147.028, Y  +743.450, Z    +0.000, E1   -53.078, E3 +42347.676}
SPL {X  -152.552, Y  +730.406, Z    +0.000, E1   -48.136, E3 +42349.093}
SPL {X  -159.377, Y  +706.804, Z    +0.000, E1   -34.828, E3 +42350.261}
SPL {X  -162.134, Y  +688.425, Z    +0.000, E1   -19.100, E3 +42350.198}
SPL {X  -162.803, Y  +675.871, Z    +0.000, E1    -5.469, E3 +42350.382}
SPL {X  -162.820, Y  +671.500, Z    +0.000, E1    +0.000, E3 +42349.950}
SPL {X  -162.820, Y  +669.743, Z    +0.000, E1    +4.352, E3 +42349.746}
SPL {X  -162.820, Y  +665.917, Z    +0.000, E1   +15.272, E3 +42349.740}
SPL {X  -162.820, Y  +661.245, Z    +0.000, E1   +28.879, E3 +42349.581}
SPL {X  -162.820, Y  +654.015, Z    +0.000, E1   +45.814, E3 +42349.728}
SPL {X  -162.820, Y  +641.345, Z    +0.000, E1   +63.138, E3 +42349.775}
SPL {X  -162.820, Y  +620.039, Z    +0.000, E1   +75.979, E3 +42348.385}
SPL {X  -162.820, Y  +571.094, Z    +0.000, E1   +77.089, E3 +42363.564}
SPL {X  -157.487, Y  +339.169, Z    +0.000, E1   +76.425, E3 +42456.668}
SPL {X  -156.386, Y  +335.181, Z    +0.000, E1   +75.555, E3 +42468.729}
SPL {X  -152.710, Y  +324.020, Z    +0.000, E1   +75.365, E3 +42476.539}
SPL {X  -139.497, Y  +296.529, Z    +0.000, E1   +77.231, E3 +42470.111}
ENDSPLINE

SPLINE
SPL {X  -139.792, Y  +297.022, Z    +0.000, E1   +76.273, E3 +42478.806}
ENDSPLINE

SPLINE
SPL {X  -138.933, Y  +295.600, Z    +0.000, E1   +75.173, E3 +42489.289}
SPL {X  -137.186, Y  +292.805, Z    +0.000, E1   +73.993, E3 +42499.879}
SPL {X  -133.270, Y  +286.961, Z    +0.000, E1   +73.739, E3 +42504.592}
SPL {X  -130.283, Y  +282.844, Z    +0.000, E1   +73.297, E3 +42509.484}
SPL {X  -126.880, Y  +278.461, Z    +0.000, E1   +72.855, E3 +42514.235}
SPL {X  -123.363, Y  +274.237, Z    +0.000, E1   +72.376, E3 +42518.717}
SPL {X  -121.018, Y  +271.573, Z    +0.000, E1   +72.049, E3 +42521.402}
SPL {X  -113.980, Y  +264.229, Z    +0.000, E1   +74.120, E3 +42516.980}
SPL {X   -56.216, Y  +227.692, Z    +0.000, E1   +56.267, E3 +42693.704}
ENDSPLINE

SPLINE
SPL {X  -126.995, Y  +278.604, Z    +0.000, E1   +59.937, E3 +42865.945}
SPL {X  -150.196, Y  +317.640, Z    +0.000, E1   +49.956, E3 +42874.400}
SPL {X  -157.261, Y  +338.316, Z    +0.000, E1   +40.017, E3 +42876.095}
SPL {X  -160.924, Y  +355.726, Z    +0.000, E1   +27.715, E3 +42876.535}
SPL {X  -162.423, Y  +369.141, Z    +0.000, E1   +15.207, E3 +42876.971}
SPL {X  -162.811, Y  +378.755, Z    +0.000, E1    +4.616, E3 +42876.885}
SPL {X  -162.820, Y  +382.684, Z    +0.000, E1    -0.227, E3 +42876.440}
SPL {X  -162.820, Y  +387.227, Z    +0.000, E1   -12.320, E3 +42876.195}
SPL {X  -162.820, Y  +392.558, Z    +0.000, E1   -27.778, E3 +42876.231}
SPL {X  -162.820, Y  +398.468, Z    +0.000, E1   -42.446, E3 +42876.081}
SPL {X  -162.820, Y  +404.415, Z    +0.000, E1   -53.236, E3 +42876.121}
SPL {X  -162.820, Y  +414.510, Z    +0.000, E1   -65.115, E3 +42875.538}
SPL {X  -162.820, Y  +465.064, Z    +0.000, E1   -76.269, E3 +42885.386}
SPL {X  -157.184, Y  +715.968, Z    +0.000, E1   -76.600, E3 +42981.343}
SPL {X  -156.461, Y  +718.560, Z    +0.000, E1   -75.553, E3 +42994.763}
SPL {X  -151.911, Y  +732.096, Z    +0.000, E1   -75.235, E3 +43005.317}
SPL {X  -146.569, Y  +744.407, Z    +0.000, E1   -74.677, E3 +43017.121}
SPL {X  -142.375, Y  +752.491, Z    +0.000, E1   -74.335, E3 +43024.149}
SPL {X  -139.539, Y  +757.399, Z    +0.000, E1   -73.892, E3 +43030.346}
SPL {X  -136.017, Y  +762.997, Z    +0.000, E1   -73.579, E3 +43035.529}
SPL {X  -133.089, Y  +767.296, Z    +0.000, E1   -73.251, E3 +43039.987}
SPL {X  -129.985, Y  +771.553, Z    +0.000, E1   -72.801, E3 +43044.981}
SPL {X  -126.581, Y  +775.909, Z    +0.000, E1   -72.426, E3 +43049.292}
SPL {X  -123.329, Y  +779.803, Z    +0.000, E1   -71.936, E3 +43053.674}
SPL {X  -119.291, Y  +784.315, Z    +0.000, E1   -72.148, E3 +43055.085}
SPL {X   -57.587, Y  +825.796, Z    +0.000, E1   -56.753, E3 +43208.848}
ENDSPLINE

SPLINE
SPL {X  -124.075, Y  +778.932, Z    +0.000, E1   -61.393, E3 +43402.477}
SPL {X  -147.028, Y  +743.450, Z    +0.000, E1   -53.078, E3 +43409.214}
SPL {X  -152.552, Y  +730.406, Z    +0.000, E1   -48.136, E3 +43410.632}
SPL {X  -159.377, Y  +706.804, Z    +0.000, E1   -34.828, E3 +43411.800}
SPL {X  -162.134, Y  +688.425, Z    +0.000, E1   -19.100, E3 +43411.736}
SPL {X  -162.803, Y  +675.871, Z    +0.000, E1    -5.469, E3 +43411.920}
SPL {X  -162.820, Y  +671.500, Z    +0.000, E1    +0.000, E3 +43411.488}
SPL {X  -162.820, Y  +669.743, Z    +0.000, E1    +4.352, E3 +43411.284}
SPL {X  -162.820, Y  +665.917, Z    +0.000, E1   +15.272, E3 +43411.279}
SPL {X  -162.820, Y  +661.245, Z    +0.000, E1   +28.879, E3 +43411.120}
SPL {X  -162.820, Y  +654.015, Z    +0.000, E1   +45.814, E3 +43411.267}
SPL {X  -162.820, Y  +641.345, Z    +0.000, E1   +63.138, E3 +43411.314}
SPL {X  -162.820, Y  +620.039, Z    +0.000, E1   +75.979, E3 +43409.924}
SPL {X  -162.820, Y  +571.094, Z    +0.000, E1   +77.089, E3 +43425.102}
SPL {X  -158.110, Y  +341.619, Z    +0.000, E1   +77.339, E3 +43506.752}
SPL {X  -156.597, Y  +335.917, Z    +0.000, E1   +75.680, E3 +43528.595}
SPL {X  -152.710, Y  +324.020, Z    +0.000, E1   +75.365, E3 +43538.077}
SPL {X  -139.497, Y  +296.529, Z    +0.000, E1   +77.231, E3 +43531.649}
ENDSPLINE

SPLINE
SPL {X  -139.792, Y  +297.022, Z    +0.000, E1   +76.273, E3 +43540.344}
ENDSPLINE

SPLINE
SPL {X  -138.933, Y  +295.600, Z    +0.000, E1   +75.173, E3 +43550.827}
SPL {X  -137.186, Y  +292.805, Z    +0.000, E1   +73.993, E3 +43561.417}
SPL {X  -133.270, Y  +286.961, Z    +0.000, E1   +73.739, E3 +43566.131}
SPL {X  -130.283, Y  +282.844, Z    +0.000, E1   +73.297, E3 +43571.023}
SPL {X  -127.795, Y  +279.610, Z    +0.000, E1   +72.860, E3 +43575.153}
SPL {X  -124.650, Y  +275.749, Z    +0.000, E1   +72.674, E3 +43578.071}
SPL {X  -121.687, Y  +272.322, Z    +0.000, E1   +72.100, E3 +43582.381}
SPL {X  -113.980, Y  +264.229, Z    +0.000, E1   +74.120, E3 +43578.519}
SPL {X   -56.216, Y  +227.692, Z    +0.000, E1   +56.267, E3 +43755.243}
ENDSPLINE

SPLINE
SPL {X  -126.995, Y  +278.604, Z    +0.000, E1   +59.937, E3 +43927.483}
SPL {X  -150.196, Y  +317.640, Z    +0.000, E1   +49.956, E3 +43935.938}
SPL {X  -157.261, Y  +338.316, Z    +0.000, E1   +40.017, E3 +43937.633}
SPL {X  -160.924, Y  +355.726, Z    +0.000, E1   +27.715, E3 +43938.074}
SPL {X  -162.423, Y  +369.141, Z    +0.000, E1   +15.207, E3 +43938.509}
SPL {X  -162.811, Y  +378.755, Z    +0.000, E1    +4.616, E3 +43938.424}
SPL {X  -162.820, Y  +382.684, Z    +0.000, E1    -0.227, E3 +43937.978}
SPL {X  -162.820, Y  +387.227, Z    +0.000, E1   -12.320, E3 +43937.733}
SPL {X  -162.820, Y  +392.558, Z    +0.000, E1   -27.778, E3 +43937.769}
SPL {X  -162.820, Y  +400.474, Z    +0.000, E1   -46.251, E3 +43937.633}
SPL {X  -162.820, Y  +414.510, Z    +0.000, E1   -65.115, E3 +43937.076}
SPL {X  -162.820, Y  +465.064, Z    +0.000, E1   -76.269, E3 +43946.924}
SPL {X  -157.184, Y  +715.968, Z    +0.000, E1   -76.600, E3 +44042.882}
SPL {X  -156.461, Y  +718.560, Z    +0.000, E1   -75.553, E3 +44056.301}
SPL {X  -151.911, Y  +732.096, Z    +0.000, E1   -75.235, E3 +44066.856}
SPL {X  -146.569, Y  +744.407, Z    +0.000, E1   -74.677, E3 +44078.660}
SPL {X  -142.375, Y  +752.491, Z    +0.000, E1   -74.335, E3 +44085.687}
SPL {X  -139.539, Y  +757.399, Z    +0.000, E1   -73.892, E3 +44091.885}
SPL {X  -136.017, Y  +762.997, Z    +0.000, E1   -73.579, E3 +44097.067}
SPL {X  -133.089, Y  +767.296, Z    +0.000, E1   -73.251, E3 +44101.525}
SPL {X  -129.985, Y  +771.553, Z    +0.000, E1   -72.801, E3 +44106.519}
SPL {X  -126.581, Y  +775.909, Z    +0.000, E1   -72.426, E3 +44110.830}
SPL {X  -123.329, Y  +779.803, Z    +0.000, E1   -71.936, E3 +44115.212}
SPL {X  -119.291, Y  +784.315, Z    +0.000, E1   -72.148, E3 +44116.624}
SPL {X   -57.587, Y  +825.796, Z    +0.000, E1   -56.753, E3 +44270.386}
ENDSPLINE

SPLINE
SPL {X  -124.075, Y  +778.932, Z    +0.000, E1   -61.393, E3 +44464.015}
SPL {X  -150.653, Y  +735.257, Z    +0.000, E1   -50.160, E3 +44471.695}
SPL {X  -159.377, Y  +706.804, Z    +0.000, E1   -34.828, E3 +44473.338}
SPL {X  -162.134, Y  +688.425, Z    +0.000, E1   -19.100, E3 +44473.275}
SPL {X  -162.803, Y  +675.871, Z    +0.000, E1    -5.469, E3 +44473.459}
SPL {X  -162.820, Y  +671.500, Z    +0.000, E1    +0.000, E3 +44473.027}
SPL {X  -162.820, Y  +669.743, Z    +0.000, E1    +4.352, E3 +44472.822}
SPL {X  -162.820, Y  +665.917, Z    +0.000, E1   +15.272, E3 +44472.817}
SPL {X  -162.820, Y  +661.245, Z    +0.000, E1   +28.879, E3 +44472.658}
SPL {X  -162.820, Y  +654.015, Z    +0.000, E1   +45.814, E3 +44472.805}
SPL {X  -162.820, Y  +641.345, Z    +0.000, E1   +63.138, E3 +44472.852}
SPL {X  -162.820, Y  +620.039, Z    +0.000, E1   +75.979, E3 +44471.462}
SPL {X  -162.820, Y  +571.094, Z    +0.000, E1   +77.089, E3 +44486.641}
SPL {X  -157.487, Y  +339.169, Z    +0.000, E1   +76.425, E3 +44579.745}
SPL {X  -156.386, Y  +335.181, Z    +0.000, E1   +75.555, E3 +44591.805}
SPL {X  -152.710, Y  +324.020, Z    +0.000, E1   +75.365, E3 +44599.616}
SPL {X  -139.497, Y  +296.529, Z    +0.000, E1   +77.231, E3 +44593.188}
ENDSPLINE

SPLINE
SPL {X  -139.792, Y  +297.022, Z    +0.000, E1   +76.273, E3 +44601.883}
ENDSPLINE

SPLINE
SPL {X  -138.933, Y  +295.600, Z    +0.000, E1   +75.173, E3 +44612.365}
SPL {X  -137.186, Y  +292.805, Z    +0.000, E1   +73.993, E3 +44622.956}
SPL {X  -133.270, Y  +286.961, Z    +0.000, E1   +73.739, E3 +44627.669}
SPL {X  -130.283, Y  +282.844, Z    +0.000, E1   +73.297, E3 +44632.561}
SPL {X  -127.795, Y  +279.610, Z    +0.000, E1   +72.860, E3 +44636.691}
SPL {X  -124.650, Y  +275.749, Z    +0.000, E1   +72.674, E3 +44639.610}
SPL {X  -121.687, Y  +272.322, Z    +0.000, E1   +72.100, E3 +44643.919}
SPL {X  -113.980, Y  +264.229, Z    +0.000, E1   +74.120, E3 +44640.057}
SPL {X   -56.216, Y  +227.692, Z    +0.000, E1   +56.267, E3 +44816.781}
ENDSPLINE

SPLINE
SPL {X  -126.995, Y  +278.604, Z    +0.000, E1   +59.937, E3 +44989.021}
SPL {X  -150.196, Y  +317.640, Z    +0.000, E1   +49.956, E3 +44997.477}
SPL {X  -157.261, Y  +338.316, Z    +0.000, E1   +40.017, E3 +44999.172}
SPL {X  -160.924, Y  +355.726, Z    +0.000, E1   +27.715, E3 +44999.612}
SPL {X  -162.423, Y  +369.141, Z    +0.000, E1   +15.207, E3 +45000.048}
SPL {X  -162.811, Y  +378.755, Z    +0.000, E1    +4.616, E3 +44999.962}
SPL {X  -162.820, Y  +382.684, Z    +0.000, E1    -0.227, E3 +44999.517}
SPL {X  -162.820, Y  +387.227, Z    +0.000, E1   -12.320, E3 +44999.272}
SPL {X  -162.820, Y  +392.558, Z    +0.000, E1   -27.778, E3 +44999.308}
SPL {X  -162.820, Y  +400.474, Z    +0.000, E1   -46.251, E3 +44999.172}
SPL {X  -162.820, Y  +414.510, Z    +0.000, E1   -65.115, E3 +44998.615}
SPL {X  -162.820, Y  +465.064, Z    +0.000, E1   -76.269, E3 +45008.463}
SPL {X  -157.184, Y  +715.968, Z    +0.000, E1   -76.600, E3 +45104.420}
SPL {X  -156.461, Y  +718.560, Z    +0.000, E1   -75.553, E3 +45117.840}
SPL {X  -151.911, Y  +732.096, Z    +0.000, E1   -75.235, E3 +45128.394}
SPL {X  -146.569, Y  +744.407, Z    +0.000, E1   -74.677, E3 +45140.198}
SPL {X  -142.375, Y  +752.491, Z    +0.000, E1   -74.335, E3 +45147.226}
SPL {X  -139.539, Y  +757.399, Z    +0.000, E1   -73.892, E3 +45153.423}
SPL {X  -136.017, Y  +762.997, Z    +0.000, E1   -73.579, E3 +45158.606}
SPL {X  -133.089, Y  +767.296, Z    +0.000, E1   -73.251, E3 +45163.064}
SPL {X  -129.985, Y  +771.553, Z    +0.000, E1   -72.801, E3 +45168.057}
SPL {X  -126.581, Y  +775.909, Z    +0.000, E1   -72.426, E3 +45172.369}
SPL {X  -123.329, Y  +779.803, Z    +0.000, E1   -71.936, E3 +45176.750}
SPL {X  -119.291, Y  +784.315, Z    +0.000, E1   -72.148, E3 +45178.162}
SPL {X   -57.587, Y  +825.796, Z    +0.000, E1   -56.753, E3 +45331.925}
ENDSPLINE

SPLINE
SPL {X  -124.075, Y  +778.932, Z    +0.000, E1   -61.393, E3 +45525.554}
SPL {X  -150.653, Y  +735.257, Z    +0.000, E1   -50.160, E3 +45533.233}
SPL {X  -159.377, Y  +706.804, Z    +0.000, E1   -34.828, E3 +45534.876}
SPL {X  -162.134, Y  +688.425, Z    +0.000, E1   -19.100, E3 +45534.813}
SPL {X  -162.803, Y  +675.871, Z    +0.000, E1    -5.469, E3 +45534.997}
SPL {X  -162.820, Y  +671.500, Z    +0.000, E1    +0.000, E3 +45534.565}
SPL {X  -162.820, Y  +669.743, Z    +0.000, E1    +4.352, E3 +45534.361}
SPL {X  -162.820, Y  +665.917, Z    +0.000, E1   +15.272, E3 +45534.355}
SPL {X  -162.820, Y  +661.245, Z    +0.000, E1   +28.879, E3 +45534.197}
SPL {X  -162.820, Y  +654.015, Z    +0.000, E1   +45.814, E3 +45534.344}
SPL {X  -162.820, Y  +641.345, Z    +0.000, E1   +63.138, E3 +45534.391}
SPL {X  -162.820, Y  +620.039, Z    +0.000, E1   +75.979, E3 +45533.001}
SPL {X  -162.820, Y  +571.094, Z    +0.000, E1   +77.089, E3 +45548.179}
SPL {X  -157.487, Y  +339.169, Z    +0.000, E1   +76.425, E3 +45641.283}
SPL {X  -156.386, Y  +335.181, Z    +0.000, E1   +75.555, E3 +45653.344}
SPL {X  -152.710, Y  +324.020, Z    +0.000, E1   +75.365, E3 +45661.154}
SPL {X  -139.497, Y  +296.529, Z    +0.000, E1   +77.231, E3 +45654.726}
ENDSPLINE

SPLINE
SPL {X  -139.792, Y  +297.022, Z    +0.000, E1   +76.273, E3 +45663.421}
ENDSPLINE

SPLINE
SPL {X  -138.933, Y  +295.600, Z    +0.000, E1   +75.173, E3 +45673.904}
SPL {X  -137.186, Y  +292.805, Z    +0.000, E1   +73.993, E3 +45684.494}
SPL {X  -133.270, Y  +286.961, Z    +0.000, E1   +73.739, E3 +45689.208}
SPL {X  -130.283, Y  +282.844, Z    +0.000, E1   +73.297, E3 +45694.100}
SPL {X  -127.795, Y  +279.610, Z    +0.000, E1   +72.860, E3 +45698.230}
SPL {X  -124.650, Y  +275.749, Z    +0.000, E1   +72.674, E3 +45701.148}
SPL {X  -121.687, Y  +272.322, Z    +0.000, E1   +72.100, E3 +45705.457}
SPL {X  -113.980, Y  +264.229, Z    +0.000, E1   +74.120, E3 +45701.596}
SPL {X   -56.216, Y  +227.692, Z    +0.000, E1   +56.267, E3 +45878.320}
ENDSPLINE

SPLINE
SPL {X  -126.995, Y  +278.604, Z    +0.000, E1   +59.937, E3 +46050.560}
SPL {X  -150.196, Y  +317.640, Z    +0.000, E1   +49.956, E3 +46059.015}
SPL {X  -157.261, Y  +338.316, Z    +0.000, E1   +40.017, E3 +46060.710}
SPL {X  -160.924, Y  +355.726, Z    +0.000, E1   +27.715, E3 +46061.151}
SPL {X  -162.423, Y  +369.141, Z    +0.000, E1   +15.207, E3 +46061.586}
SPL {X  -162.811, Y  +378.755, Z    +0.000, E1    +4.616, E3 +46061.501}
SPL {X  -162.820, Y  +382.684, Z    +0.000, E1    -0.227, E3 +46061.055}
SPL {X  -162.820, Y  +387.227, Z    +0.000, E1   -12.320, E3 +46060.810}
SPL {X  -162.820, Y  +392.558, Z    +0.000, E1   -27.778, E3 +46060.846}
SPL {X  -162.820, Y  +400.474, Z    +0.000, E1   -46.251, E3 +46060.710}
SPL {X  -162.820, Y  +414.510, Z    +0.000, E1   -65.115, E3 +46060.153}
SPL {X  -162.820, Y  +465.064, Z    +0.000, E1   -76.269, E3 +46070.001}
SPL {X  -157.184, Y  +715.968, Z    +0.000, E1   -76.600, E3 +46165.959}
SPL {X  -156.461, Y  +718.560, Z    +0.000, E1   -75.553, E3 +46179.378}
SPL {X  -151.911, Y  +732.096, Z    +0.000, E1   -75.235, E3 +46189.932}
SPL {X  -146.569, Y  +744.407, Z    +0.000, E1   -74.677, E3 +46201.737}
SPL {X  -142.375, Y  +752.491, Z    +0.000, E1   -74.335, E3 +46208.764}
SPL {X  -139.539, Y  +757.399, Z    +0.000, E1   -73.892, E3 +46214.962}
SPL {X  -136.017, Y  +762.997, Z    +0.000, E1   -73.579, E3 +46220.144}
SPL {X  -133.089, Y  +767.296, Z    +0.000, E1   -73.251, E3 +46224.602}
SPL {X  -129.985, Y  +771.553, Z    +0.000, E1   -72.801, E3 +46229.596}
SPL {X  -126.581, Y  +775.909, Z    +0.000, E1   -72.426, E3 +46233.907}
SPL {X  -123.329, Y  +779.803, Z    +0.000, E1   -71.936, E3 +46238.289}
SPL {X  -119.291, Y  +784.315, Z    +0.000, E1   -72.148, E3 +46239.701}
SPL {X   -57.587, Y  +825.796, Z    +0.000, E1   -56.753, E3 +46393.463}
ENDSPLINE

SPLINE
SPL {X  -124.075, Y  +778.932, Z    +0.000, E1   -61.393, E3 +46587.092}
SPL {X  -150.653, Y  +735.257, Z    +0.000, E1   -50.160, E3 +46594.772}
SPL {X  -159.377, Y  +706.804, Z    +0.000, E1   -34.828, E3 +46596.415}
SPL {X  -162.134, Y  +688.425, Z    +0.000, E1   -19.100, E3 +46596.352}
SPL {X  -162.803, Y  +675.871, Z    +0.000, E1    -5.469, E3 +46596.536}
SPL {X  -162.820, Y  +671.500, Z    +0.000, E1    +0.000, E3 +46596.104}
SPL {X  -162.820, Y  +669.743, Z    +0.000, E1    +4.352, E3 +46595.899}
SPL {X  -162.820, Y  +665.917, Z    +0.000, E1   +15.272, E3 +46595.894}
SPL {X  -162.820, Y  +661.245, Z    +0.000, E1   +28.879, E3 +46595.735}
SPL {X  -162.820, Y  +654.015, Z    +0.000, E1   +45.814, E3 +46595.882}
SPL {X  -162.820, Y  +641.345, Z    +0.000, E1   +63.138, E3 +46595.929}
SPL {X  -162.820, Y  +620.039, Z    +0.000, E1   +75.979, E3 +46594.539}
SPL {X  -162.820, Y  +571.094, Z    +0.000, E1   +77.089, E3 +46609.718}
SPL {X  -158.110, Y  +341.619, Z    +0.000, E1   +77.339, E3 +46691.367}
SPL {X  -156.597, Y  +335.917, Z    +0.000, E1   +75.680, E3 +46713.211}
SPL {X  -152.710, Y  +324.020, Z    +0.000, E1   +75.365, E3 +46722.693}
SPL {X  -139.497, Y  +296.529, Z    +0.000, E1   +77.231, E3 +46716.264}
ENDSPLINE

SPLINE
SPL {X  -139.792, Y  +297.022, Z    +0.000, E1   +76.273, E3 +46724.960}
ENDSPLINE

SPLINE
SPL {X  -138.933, Y  +295.600, Z    +0.000, E1   +75.173, E3 +46735.442}
SPL {X  -137.186, Y  +292.805, Z    +0.000, E1   +73.993, E3 +46746.033}
SPL {X  -133.270, Y  +286.961, Z    +0.000, E1   +73.739, E3 +46750.746}
SPL {X  -130.283, Y  +282.844, Z    +0.000, E1   +73.297, E3 +46755.638}
SPL {X  -127.795, Y  +279.610, Z    +0.000, E1   +72.860, E3 +46759.768}
SPL {X  -124.650, Y  +275.749, Z    +0.000, E1   +72.674, E3 +46762.687}
SPL {X  -121.687, Y  +272.322, Z    +0.000, E1   +72.100, E3 +46766.996}
SPL {X  -113.980, Y  +264.229, Z    +0.000, E1   +74.120, E3 +46763.134}
SPL {X   -56.216, Y  +227.692, Z    +0.000, E1   +56.267, E3 +46939.858}
ENDSPLINE

SPLINE
SPL {X  -126.995, Y  +278.604, Z    +0.000, E1   +59.937, E3 +47112.098}
SPL {X  -150.196, Y  +317.640, Z    +0.000, E1   +49.956, E3 +47120.553}
SPL {X  -157.261, Y  +338.316, Z    +0.000, E1   +40.017, E3 +47122.249}
SPL {X  -160.924, Y  +355.726, Z    +0.000, E1   +27.715, E3 +47122.689}
SPL {X  -162.423, Y  +369.141, Z    +0.000, E1   +15.207, E3 +47123.125}
SPL {X  -162.811, Y  +378.755, Z    +0.000, E1    +4.616, E3 +47123.039}
SPL {X  -162.820, Y  +382.684, Z    +0.000, E1    -0.227, E3 +47122.594}
SPL {X  -162.820, Y  +385.721, Z    +0.000, E1    -8.371, E3 +47122.409}
SPL {X  -162.820, Y  +388.532, Z    +0.000, E1   -16.412, E3 +47122.296}
SPL {X  -162.820, Y  +392.558, Z    +0.000, E1   -27.778, E3 +47122.385}
SPL {X  -162.820, Y  +400.474, Z    +0.000, E1   -46.251, E3 +47122.248}
SPL {X  -162.820, Y  +414.510, Z    +0.000, E1   -65.115, E3 +47121.692}
SPL {X  -162.820, Y  +465.064, Z    +0.000, E1   -76.269, E3 +47131.540}
SPL {X  -158.097, Y  +712.432, Z    +0.000, E1   -77.677, E3 +47213.927}
SPL {X  -156.557, Y  +718.224, Z    +0.000, E1   -75.715, E3 +47239.064}
SPL {X  -153.015, Y  +729.150, Z    +0.000, E1   -75.312, E3 +47249.006}
SPL {X  -149.053, Y  +739.025, Z    +0.000, E1   -74.952, E3 +47257.802}
SPL {X  -145.525, Y  +746.527, Z    +0.000, E1   -74.526, E3 +47265.595}
SPL {X  -142.375, Y  +752.491, Z    +0.000, E1   -74.335, E3 +47270.303}
SPL {X  -139.539, Y  +757.399, Z    +0.000, E1   -73.892, E3 +47276.500}
SPL {X  -136.017, Y  +762.997, Z    +0.000, E1   -73.579, E3 +47281.683}
SPL {X  -133.089, Y  +767.296, Z    +0.000, E1   -73.251, E3 +47286.141}
SPL {X  -129.985, Y  +771.553, Z    +0.000, E1   -72.801, E3 +47291.134}
SPL {X  -126.581, Y  +775.909, Z    +0.000, E1   -72.426, E3 +47295.446}
SPL {X  -123.329, Y  +779.803, Z    +0.000, E1   -71.936, E3 +47299.827}
SPL {X  -119.291, Y  +784.315, Z    +0.000, E1   -72.148, E3 +47301.239}
SPL {X   -57.587, Y  +825.796, Z    +0.000, E1   -56.753, E3 +47455.002}
ENDSPLINE

SPLINE
SPL {X  -124.075, Y  +778.932, Z    +0.000, E1   -61.393, E3 +47648.631}
SPL {X  -150.653, Y  +735.257, Z    +0.000, E1   -50.160, E3 +47656.310}
SPL {X  -159.377, Y  +706.804, Z    +0.000, E1   -34.828, E3 +47657.953}
SPL {X  -162.134, Y  +688.425, Z    +0.000, E1   -19.100, E3 +47657.890}
SPL {X  -162.803, Y  +675.871, Z    +0.000, E1    -5.469, E3 +47658.074}
SPL {X  -162.820, Y  +671.500, Z    +0.000, E1    +0.000, E3 +47657.642}
SPL {X  -162.820, Y  +669.743, Z    +0.000, E1    +4.352, E3 +47657.438}
SPL {X  -162.820, Y  +665.917, Z    +0.000, E1   +15.272, E3 +47657.432}
SPL {X  -162.820, Y  +659.880, Z    +0.000, E1   +32.256, E3 +47657.344}
SPL {X  -162.820, Y  +652.069, Z    +0.000, E1   +49.663, E3 +47657.369}
SPL {X  -162.820, Y  +641.345, Z    +0.000, E1   +63.138, E3 +47657.468}
SPL {X  -162.820, Y  +620.039, Z    +0.000, E1   +75.979, E3 +47656.078}
SPL {X  -162.820, Y  +571.094, Z    +0.000, E1   +77.089, E3 +47671.256}
SPL {X  -157.487, Y  +339.169, Z    +0.000, E1   +76.425, E3 +47764.360}
SPL {X  -156.386, Y  +335.181, Z    +0.000, E1   +75.555, E3 +47776.421}
SPL {X  -152.710, Y  +324.020, Z    +0.000, E1   +75.365, E3 +47784.231}
SPL {X  -139.497, Y  +296.529, Z    +0.000, E1   +77.231, E3 +47777.803}
ENDSPLINE

SPLINE
SPL {X  -139.792, Y  +297.022, Z    +0.000, E1   +76.273, E3 +47786.498}
ENDSPLINE

SPLINE
SPL {X  -138.933, Y  +295.600, Z    +0.000, E1   +75.173, E3 +47796.981}
SPL {X  -137.186, Y  +292.805, Z    +0.000, E1   +73.993, E3 +47807.571}
SPL {X  -133.270, Y  +286.961, Z    +0.000, E1   +73.739, E3 +47812.285}
SPL {X  -129.057, Y  +281.230, Z    +0.000, E1   +73.118, E3 +47819.192}
SPL {X  -123.859, Y  +274.815, Z    +0.000, E1   +72.511, E3 +47825.577}
SPL {X  -121.018, Y  +271.573, Z    +0.000, E1   +72.049, E3 +47829.094}
SPL {X  -113.980, Y  +264.229, Z    +0.000, E1   +74.120, E3 +47824.673}
SPL {X   -56.216, Y  +227.692, Z    +0.000, E1   +56.267, E3 +48001.397}
ENDSPLINE

SPLINE
SPL {X  -126.995, Y  +278.604, Z    +0.000, E1   +59.937, E3 +48173.637}
SPL {X  -150.196, Y  +317.640, Z    +0.000, E1   +49.956, E3 +48182.092}
SPL {X  -157.261, Y  +338.316, Z    +0.000, E1   +40.017, E3 +48183.787}
SPL {X  -160.924, Y  +355.726, Z    +0.000, E1   +27.715, E3 +48184.228}
SPL {X  -162.423, Y  +369.141, Z    +0.000, E1   +15.207, E3 +48184.663}
SPL {X  -162.811, Y  +378.755, Z    +0.000, E1    +4.616, E3 +48184.578}
SPL {X  -162.820, Y  +382.684, Z    +0.000, E1    -0.227, E3 +48184.132}
SPL {X  -162.820, Y  +385.721, Z    +0.000, E1    -8.371, E3 +48183.948}
SPL {X  -162.820, Y  +388.532, Z    +0.000, E1   -16.412, E3 +48183.834}
SPL {X  -162.820, Y  +392.558, Z    +0.000, E1   -27.778, E3 +48183.923}
SPL {X  -162.820, Y  +398.468, Z    +0.000, E1   -42.446, E3 +48183.774}
SPL {X  -162.820, Y  +404.415, Z    +0.000, E1   -53.236, E3 +48183.813}
SPL {X  -162.820, Y  +414.510, Z    +0.000, E1   -65.115, E3 +48183.230}
SPL {X  -162.820, Y  +457.766, Z    +0.000, E1   -75.929, E3 +48191.066}
SPL {X  -162.820, Y  +471.144, Z    +0.000, E1   -76.496, E3 +48194.755}
SPL {X  -158.097, Y  +712.432, Z    +0.000, E1   -77.677, E3 +48275.466}
SPL {X  -156.557, Y  +718.224, Z    +0.000, E1   -75.715, E3 +48300.602}
SPL {X  -153.015, Y  +729.150, Z    +0.000, E1   -75.312, E3 +48310.544}
SPL {X  -149.053, Y  +739.025, Z    +0.000, E1   -74.952, E3 +48319.340}
SPL {X  -144.053, Y  +749.389, Z    +0.000, E1   -74.457, E3 +48329.332}
SPL {X  -139.539, Y  +757.399, Z    +0.000, E1   -73.892, E3 +48338.039}
SPL {X  -136.017, Y  +762.997, Z    +0.000, E1   -73.579, E3 +48343.221}
SPL {X  -133.089, Y  +767.296, Z    +0.000, E1   -73.251, E3 +48347.679}
SPL {X  -129.985, Y  +771.553, Z    +0.000, E1   -72.801, E3 +48352.673}
SPL {X  -126.581, Y  +775.909, Z    +0.000, E1   -72.426, E3 +48356.984}
SPL {X  -123.329, Y  +779.803, Z    +0.000, E1   -71.936, E3 +48361.366}
SPL {X  -119.291, Y  +784.315, Z    +0.000, E1   -72.148, E3 +48362.778}
SPL {X   -57.587, Y  +825.796, Z    +0.000, E1   -56.753, E3 +48516.540}
ENDSPLINE

SPLINE
SPL {X  -124.075, Y  +778.932, Z    +0.000, E1   -61.393, E3 +48710.169}
SPL {X  -150.653, Y  +735.257, Z    +0.000, E1   -50.160, E3 +48717.848}
SPL {X  -159.377, Y  +706.804, Z    +0.000, E1   -34.828, E3 +48719.492}
SPL {X  -162.134, Y  +688.425, Z    +0.000, E1   -19.100, E3 +48719.429}
SPL {X  -162.803, Y  +675.871, Z    +0.000, E1    -5.469, E3 +48719.613}
SPL {X  -162.820, Y  +671.500, Z    +0.000, E1    +0.000, E3 +48719.181}
SPL {X  -162.820, Y  +669.743, Z    +0.000, E1    +4.352, E3 +48718.976}
SPL {X  -162.820, Y  +665.917, Z    +0.000, E1   +15.272, E3 +48718.971}
SPL {X  -162.820, Y  +661.245, Z    +0.000, E1   +28.879, E3 +48718.812}
SPL {X  -162.820, Y  +654.015, Z    +0.000, E1   +45.814, E3 +48718.959}
SPL {X  -162.820, Y  +641.345, Z    +0.000, E1   +63.138, E3 +48719.006}
SPL {X  -162.820, Y  +620.039, Z    +0.000, E1   +75.979, E3 +48717.616}
SPL {X  -162.820, Y  +571.094, Z    +0.000, E1   +77.089, E3 +48732.795}
SPL {X  -157.487, Y  +339.169, Z    +0.000, E1   +76.425, E3 +48825.898}
SPL {X  -156.386, Y  +335.181, Z    +0.000, E1   +75.555, E3 +48837.959}
SPL {X  -152.710, Y  +324.020, Z    +0.000, E1   +75.365, E3 +48845.770}
SPL {X  -139.497, Y  +296.529, Z    +0.000, E1   +77.231, E3 +48839.341}
ENDSPLINE

SPLINE
SPL {X  -139.792, Y  +297.022, Z    +0.000, E1   +76.273, E3 +48848.037}
ENDSPLINE

SPLINE
SPL {X  -138.933, Y  +295.600, Z    +0.000, E1   +75.173, E3 +48858.519}
SPL {X  -137.186, Y  +292.805, Z    +0.000, E1   +73.993, E3 +48869.110}
SPL {X  -133.270, Y  +286.961, Z    +0.000, E1   +73.739, E3 +48873.823}
SPL {X  -130.283, Y  +282.844, Z    +0.000, E1   +73.297, E3 +48878.715}
SPL {X  -126.880, Y  +278.461, Z    +0.000, E1   +72.855, E3 +48883.466}
SPL {X  -123.363, Y  +274.237, Z    +0.000, E1   +72.376, E3 +48887.948}
SPL {X  -121.018, Y  +271.573, Z    +0.000, E1   +72.049, E3 +48890.633}
SPL {X  -113.980, Y  +264.229, Z    +0.000, E1   +74.120, E3 +48886.211}
SPL {X   -56.216, Y  +227.692, Z    +0.000, E1   +56.267, E3 +49062.935}
ENDSPLINE

SPLINE
SPL {X  -126.995, Y  +278.604, Z    +0.000, E1   +59.937, E3 +49235.175}
SPL {X  -150.196, Y  +317.640, Z    +0.000, E1   +49.956, E3 +49243.630}
SPL {X  -157.261, Y  +338.316, Z    +0.000, E1   +40.017, E3 +49245.326}
SPL {X  -160.924, Y  +355.726, Z    +0.000, E1   +27.715, E3 +49245.766}
SPL {X  -162.423, Y  +369.141, Z    +0.000, E1   +15.207, E3 +49246.202}
SPL {X  -162.811, Y  +378.755, Z    +0.000, E1    +4.616, E3 +49246.116}
SPL {X  -162.820, Y  +382.684, Z    +0.000, E1    -0.227, E3 +49245.671}
SPL {X  -162.820, Y  +387.227, Z    +0.000, E1   -12.320, E3 +49245.426}
SPL {X  -162.820, Y  +392.558, Z    +0.000, E1   -27.778, E3 +49245.462}
SPL {X  -162.820, Y  +400.474, Z    +0.000, E1   -46.251, E3 +49245.325}
SPL {X  -162.820, Y  +414.510, Z    +0.000, E1   -65.115, E3 +49244.769}
SPL {X  -162.820, Y  +457.766, Z    +0.000, E1   -75.929, E3 +49252.605}
SPL {X  -162.820, Y  +471.144, Z    +0.000, E1   -76.496, E3 +49256.294}
SPL {X  -158.097, Y  +712.432, Z    +0.000, E1   -77.677, E3 +49337.004}
SPL {X  -156.557, Y  +718.224, Z    +0.000, E1   -75.715, E3 +49362.141}
SPL {X  -151.911, Y  +732.096, Z    +0.000, E1   -75.235, E3 +49374.548}
SPL {X  -146.569, Y  +744.407, Z    +0.000, E1   -74.677, E3 +49386.352}
SPL {X  -142.375, Y  +752.491, Z    +0.000, E1   -74.335, E3 +49393.379}
SPL {X  -139.539, Y  +757.399, Z    +0.000, E1   -73.892, E3 +49399.577}
SPL {X  -136.017, Y  +762.997, Z    +0.000, E1   -73.579, E3 +49404.759}
SPL {X  -133.089, Y  +767.296, Z    +0.000, E1   -73.251, E3 +49409.218}
SPL {X  -129.985, Y  +771.553, Z    +0.000, E1   -72.801, E3 +49414.211}
SPL {X  -126.581, Y  +775.909, Z    +0.000, E1   -72.426, E3 +49418.522}
SPL {X  -123.329, Y  +779.803, Z    +0.000, E1   -71.936, E3 +49422.904}
SPL {X  -119.291, Y  +784.315, Z    +0.000, E1   -72.148, E3 +49424.316}
SPL {X   -57.587, Y  +825.796, Z    +0.000, E1   -56.753, E3 +49578.079}
ENDSPLINE

SPLINE
SPL {X  -124.075, Y  +778.932, Z    +0.000, E1   -61.393, E3 +49771.708}
SPL {X  -150.653, Y  +735.257, Z    +0.000, E1   -50.160, E3 +49779.387}
SPL {X  -159.377, Y  +706.804, Z    +0.000, E1   -34.828, E3 +49781.030}
SPL {X  -162.134, Y  +688.425, Z    +0.000, E1   -19.100, E3 +49780.967}
SPL {X  -162.734, Y  +678.779, Z    +0.000, E1    -8.745, E3 +49781.106}
SPL {X  -162.820, Y  +671.589, Z    +0.000, E1    -0.221, E3 +49780.741}
SPL {X  -162.820, Y  +669.743, Z    +0.000, E1    +4.352, E3 +49780.515}
SPL {X  -162.820, Y  +665.917, Z    +0.000, E1   +15.272, E3 +49780.509}
SPL {X  -162.820, Y  +659.880, Z    +0.000, E1   +32.256, E3 +49780.421}
SPL {X  -162.820, Y  +652.069, Z    +0.000, E1   +49.663, E3 +49780.446}
SPL {X  -162.820, Y  +641.345, Z    +0.000, E1   +63.138, E3 +49780.545}
SPL {X  -162.820, Y  +620.039, Z    +0.000, E1   +75.979, E3 +49779.154}
SPL {X  -162.820, Y  +571.094, Z    +0.000, E1   +77.089, E3 +49794.333}
SPL {X  -158.110, Y  +341.619, Z    +0.000, E1   +77.339, E3 +49875.983}
SPL {X  -156.597, Y  +335.917, Z    +0.000, E1   +75.680, E3 +49897.826}
SPL {X  -152.710, Y  +324.020, Z    +0.000, E1   +75.365, E3 +49907.308}
SPL {X  -139.497, Y  +296.529, Z    +0.000, E1   +77.231, E3 +49900.880}
ENDSPLINE

SPLINE
SPL {X  -139.792, Y  +297.022, Z    +0.000, E1   +76.273, E3 +49909.575}
ENDSPLINE

SPLINE
SPL {X  -138.933, Y  +295.600, Z    +0.000, E1   +75.173, E3 +49920.058}
SPL {X  -137.186, Y  +292.805, Z    +0.000, E1   +73.993, E3 +49930.648}
SPL {X  -133.270, Y  +286.961, Z    +0.000, E1   +73.739, E3 +49935.362}
SPL {X  -130.283, Y  +282.844, Z    +0.000, E1   +73.297, E3 +49940.253}
SPL {X  -126.880, Y  +278.461, Z    +0.000, E1   +72.855, E3 +49945.004}
SPL {X  -123.363, Y  +274.237, Z    +0.000, E1   +72.376, E3 +49949.486}
SPL {X  -121.018, Y  +271.573, Z    +0.000, E1   +72.049, E3 +49952.171}
SPL {X  -113.980, Y  +264.229, Z    +0.000, E1   +74.120, E3 +49947.750}
SPL {X   -56.216, Y  +227.692, Z    +0.000, E1   +56.267, E3 +50124.474}
ENDSPLINE

SPLINE
SPL {X  -126.995, Y  +278.604, Z    +0.000, E1   +59.937, E3 +50296.714}
SPL {X  -150.196, Y  +317.640, Z    +0.000, E1   +49.956, E3 +50305.169}
SPL {X  -157.261, Y  +338.316, Z    +0.000, E1   +40.017, E3 +50306.864}
SPL {X  -160.924, Y  +355.726, Z    +0.000, E1   +27.715, E3 +50307.305}
SPL {X  -162.423, Y  +369.141, Z    +0.000, E1   +15.207, E3 +50307.740}
SPL {X  -162.811, Y  +378.755, Z    +0.000, E1    +4.616, E3 +50307.655}
SPL {X  -162.820, Y  +382.684, Z    +0.000, E1    -0.227, E3 +50307.209}
SPL {X  -162.820, Y  +385.721, Z    +0.000, E1    -8.371, E3 +50307.025}
SPL {X  -162.820, Y  +388.532, Z    +0.000, E1   -16.412, E3 +50306.911}
SPL {X  -162.820, Y  +392.558, Z    +0.000, E1   -27.778, E3 +50307.000}
SPL {X  -162.820, Y  +400.474, Z    +0.000, E1   -46.251, E3 +50306.864}
SPL {X  -162.820, Y  +414.510, Z    +0.000, E1   -65.115, E3 +50306.307}
SPL {X  -162.820, Y  +465.064, Z    +0.000, E1   -76.269, E3 +50316.155}
SPL {X  -157.184, Y  +715.968, Z    +0.000, E1   -76.600, E3 +50412.112}
SPL {X  -156.461, Y  +718.560, Z    +0.000, E1   -75.553, E3 +50425.532}
SPL {X  -151.911, Y  +732.096, Z    +0.000, E1   -75.235, E3 +50436.086}
SPL {X  -146.569, Y  +744.407, Z    +0.000, E1   -74.677, E3 +50447.891}
SPL {X  -142.375, Y  +752.491, Z    +0.000, E1   -74.335, E3 +50454.918}
SPL {X  -139.539, Y  +757.399, Z    +0.000, E1   -73.892, E3 +50461.116}
SPL {X  -136.017, Y  +762.997, Z    +0.000, E1   -73.579, E3 +50466.298}
SPL {X  -133.089, Y  +767.296, Z    +0.000, E1   -73.251, E3 +50470.756}
SPL {X  -129.985, Y  +771.553, Z    +0.000, E1   -72.801, E3 +50475.750}
SPL {X  -126.581, Y  +775.909, Z    +0.000, E1   -72.426, E3 +50480.061}
SPL {X  -122.528, Y  +780.725, Z    +0.000, E1   -71.905, E3 +50485.081}
SPL {X  -116.189, Y  +787.563, Z    +0.000, E1   -72.978, E3 +50484.365}
SPL {X   -57.587, Y  +825.796, Z    +0.000, E1   -56.753, E3 +50639.617}
ENDSPLINE

SPLINE
SPL {X  -124.075, Y  +778.932, Z    +0.000, E1   -61.393, E3 +50833.246}
SPL {X  -147.028, Y  +743.450, Z    +0.000, E1   -53.078, E3 +50839.983}
SPL {X  -152.552, Y  +730.406, Z    +0.000, E1   -48.136, E3 +50841.401}
SPL {X  -159.377, Y  +706.804, Z    +0.000, E1   -34.828, E3 +50842.569}
SPL {X  -162.134, Y  +688.425, Z    +0.000, E1   -19.100, E3 +50842.506}
SPL {X  -162.803, Y  +675.871, Z    +0.000, E1    -5.469, E3 +50842.690}
SPL {X  -162.820, Y  +671.500, Z    +0.000, E1    +0.000, E3 +50842.258}
SPL {X  -162.820, Y  +669.743, Z    +0.000, E1    +4.352, E3 +50842.053}
SPL {X  -162.820, Y  +665.917, Z    +0.000, E1   +15.272, E3 +50842.048}
SPL {X  -162.820, Y  +661.245, Z    +0.000, E1   +28.879, E3 +50841.889}
SPL {X  -162.820, Y  +654.015, Z    +0.000, E1   +45.814, E3 +50842.036}
SPL {X  -162.820, Y  +641.345, Z    +0.000, E1   +63.138, E3 +50842.083}
SPL {X  -162.820, Y  +620.039, Z    +0.000, E1   +75.979, E3 +50840.693}
SPL {X  -162.820, Y  +571.094, Z    +0.000, E1   +77.089, E3 +50855.872}
SPL {X  -157.487, Y  +339.169, Z    +0.000, E1   +76.425, E3 +50948.975}
SPL {X  -156.386, Y  +335.181, Z    +0.000, E1   +75.555, E3 +50961.036}
SPL {X  -152.710, Y  +324.020, Z    +0.000, E1   +75.365, E3 +50968.847}
SPL {X  -139.497, Y  +296.529, Z    +0.000, E1   +77.231, E3 +50962.418}
ENDSPLINE

SPLINE
SPL {X  -139.520, Y  +296.568, Z    +0.000, E1   +75.884, E3 +50975.066}
ENDSPLINE

SPLINE
SPL {X  -138.554, Y  +294.984, Z    +0.000, E1   +74.772, E3 +50984.947}
SPL {X  -137.186, Y  +292.805, Z    +0.000, E1   +73.993, E3 +50992.187}
SPL {X  -133.270, Y  +286.961, Z    +0.000, E1   +73.739, E3 +50996.900}
SPL {X  -130.283, Y  +282.844, Z    +0.000, E1   +73.297, E3 +51001.792}
SPL {X  -127.795, Y  +279.610, Z    +0.000, E1   +72.860, E3 +51005.922}
SPL {X  -124.650, Y  +275.749, Z    +0.000, E1   +72.674, E3 +51008.840}
SPL {X  -121.687, Y  +272.322, Z    +0.000, E1   +72.100, E3 +51013.150}
SPL {X  -113.980, Y  +264.229, Z    +0.000, E1   +74.120, E3 +51009.288}
SPL {X   -56.216, Y  +227.692, Z    +0.000, E1   +56.267, E3 +51186.012}
ENDSPLINE

SPLINE
SPL {X  -126.995, Y  +278.604, Z    +0.000, E1   +59.937, E3 +51358.252}
SPL {X  -150.196, Y  +317.640, Z    +0.000, E1   +49.956, E3 +51366.707}
SPL {X  -157.261, Y  +338.316, Z    +0.000, E1   +40.017, E3 +51368.402}
SPL {X  -160.924, Y  +355.726, Z    +0.000, E1   +27.715, E3 +51368.843}
SPL {X  -162.423, Y  +369.141, Z    +0.000, E1   +15.207, E3 +51369.279}
SPL {X  -162.811, Y  +378.755, Z    +0.000, E1    +4.616, E3 +51369.193}
SPL {X  -162.820, Y  +382.684, Z    +0.000, E1    -0.227, E3 +51368.748}
SPL {X  -162.820, Y  +387.227, Z    +0.000, E1   -12.320, E3 +51368.502}
SPL {X  -162.820, Y  +392.558, Z    +0.000, E1   -27.778, E3 +51368.539}
SPL {X  -162.820, Y  +400.474, Z    +0.000, E1   -46.251, E3 +51368.402}
SPL {X  -162.820, Y  +414.510, Z    +0.000, E1   -65.115, E3 +51367.845}
SPL {X  -162.820, Y  +465.064, Z    +0.000, E1   -76.269, E3 +51377.693}
SPL {X  -157.184, Y  +715.968, Z    +0.000, E1   -76.600, E3 +51473.651}
SPL {X  -156.461, Y  +718.560, Z    +0.000, E1   -75.553, E3 +51487.071}
SPL {X  -151.911, Y  +732.096, Z    +0.000, E1   -75.235, E3 +51497.625}
SPL {X  -146.569, Y  +744.407, Z    +0.000, E1   -74.677, E3 +51509.429}
SPL {X  -142.375, Y  +752.491, Z    +0.000, E1   -74.335, E3 +51516.456}
SPL {X  -139.539, Y  +757.399, Z    +0.000, E1   -73.892, E3 +51522.654}
SPL {X  -136.017, Y  +762.997, Z    +0.000, E1   -73.579, E3 +51527.836}
SPL {X  -133.089, Y  +767.296, Z    +0.000, E1   -73.251, E3 +51532.294}
SPL {X  -129.985, Y  +771.553, Z    +0.000, E1   -72.801, E3 +51537.288}
SPL {X  -126.581, Y  +775.909, Z    +0.000, E1   -72.426, E3 +51541.599}
SPL {X  -123.329, Y  +779.803, Z    +0.000, E1   -71.936, E3 +51545.981}
SPL {X  -119.291, Y  +784.315, Z    +0.000, E1   -72.148, E3 +51547.393}
SPL {X   -57.587, Y  +825.796, Z    +0.000, E1   -56.753, E3 +51701.156}
ENDSPLINE

SPLINE
SPL {X  -124.075, Y  +778.932, Z    +0.000, E1   -61.393, E3 +51894.785}
SPL {X  -150.653, Y  +735.257, Z    +0.000, E1   -50.160, E3 +51902.464}
SPL {X  -159.377, Y  +706.804, Z    +0.000, E1   -34.828, E3 +51904.107}
SPL {X  -162.134, Y  +688.425, Z    +0.000, E1   -19.100, E3 +51904.044}
SPL {X  -162.803, Y  +675.871, Z    +0.000, E1    -5.469, E3 +51904.228}
SPL {X  -162.820, Y  +671.500, Z    +0.000, E1    +0.000, E3 +51903.796}
SPL {X  -162.820, Y  +669.743, Z    +0.000, E1    +4.352, E3 +51903.592}
SPL {X  -162.820, Y  +665.917, Z    +0.000, E1   +15.272, E3 +51903.586}
SPL {X  -162.820, Y  +661.245, Z    +0.000, E1   +28.879, E3 +51903.427}
SPL {X  -162.820, Y  +654.015, Z    +0.000, E1   +45.814, E3 +51903.574}
SPL {X  -162.820, Y  +641.345, Z    +0.000, E1   +63.138, E3 +51903.622}
SPL {X  -162.820, Y  +620.039, Z    +0.000, E1   +75.979, E3 +51902.231}
SPL {X  -162.820, Y  +571.094, Z    +0.000, E1   +77.089, E3 +51917.410}
SPL {X  -157.487, Y  +339.169, Z    +0.000, E1   +76.425, E3 +52010.514}
SPL {X  -156.386, Y  +335.181, Z    +0.000, E1   +75.555, E3 +52022.575}
SPL {X  -152.710, Y  +324.020, Z    +0.000, E1   +75.365, E3 +52030.385}
SPL {X  -139.497, Y  +296.529, Z    +0.000, E1   +77.231, E3 +52023.957}
ENDSPLINE

SPLINE
SPL {X  -139.792, Y  +297.022, Z    +0.000, E1   +76.273, E3 +52032.652}
ENDSPLINE

SPLINE
SPL {X  -138.933, Y  +295.600, Z    +0.000, E1   +75.173, E3 +52043.135}
SPL {X  -137.186, Y  +292.805, Z    +0.000, E1   +73.993, E3 +52053.725}
SPL {X  -133.270, Y  +286.961, Z    +0.000, E1   +73.739, E3 +52058.438}
SPL {X  -130.283, Y  +282.844, Z    +0.000, E1   +73.297, E3 +52063.330}
SPL {X  -127.795, Y  +279.610, Z    +0.000, E1   +72.860, E3 +52067.461}
SPL {X  -124.650, Y  +275.749, Z    +0.000, E1   +72.674, E3 +52070.379}
SPL {X  -121.687, Y  +272.322, Z    +0.000, E1   +72.100, E3 +52074.688}
SPL {X  -113.980, Y  +264.229, Z    +0.000, E1   +74.120, E3 +52070.826}
SPL {X   -56.216, Y  +227.692, Z    +0.000, E1   +56.267, E3 +52247.550}
ENDSPLINE

SPLINE
SPL {X  -126.995, Y  +278.604, Z    +0.000, E1   +59.937, E3 +52419.791}
SPL {X  -150.196, Y  +317.640, Z    +0.000, E1   +49.956, E3 +52428.246}
SPL {X  -157.261, Y  +338.316, Z    +0.000, E1   +40.017, E3 +52429.941}
SPL {X  -160.924, Y  +355.726, Z    +0.000, E1   +27.715, E3 +52430.382}
SPL {X  -162.423, Y  +369.141, Z    +0.000, E1   +15.207, E3 +52430.817}
SPL {X  -162.811, Y  +378.755, Z    +0.000, E1    +4.616, E3 +52430.732}
SPL {X  -162.820, Y  +382.684, Z    +0.000, E1    -0.227, E3 +52430.286}
SPL {X  -162.820, Y  +387.227, Z    +0.000, E1   -12.320, E3 +52430.041}
SPL {X  -162.820, Y  +392.558, Z    +0.000, E1   -27.778, E3 +52430.077}
SPL {X  -162.820, Y  +400.474, Z    +0.000, E1   -46.251, E3 +52429.941}
SPL {X  -162.820, Y  +414.510, Z    +0.000, E1   -65.115, E3 +52429.384}
SPL {X  -162.820, Y  +465.064, Z    +0.000, E1   -76.269, E3 +52439.232}
SPL {X  -157.184, Y  +715.968, Z    +0.000, E1   -76.600, E3 +52535.189}
SPL {X  -156.461, Y  +718.560, Z    +0.000, E1   -75.553, E3 +52548.609}
SPL {X  -153.015, Y  +729.150, Z    +0.000, E1   -75.312, E3 +52556.698}
SPL {X  -149.053, Y  +739.025, Z    +0.000, E1   -74.952, E3 +52565.494}
SPL {X  -145.525, Y  +746.527, Z    +0.000, E1   -74.526, E3 +52573.287}
SPL {X  -142.375, Y  +752.491, Z    +0.000, E1   -74.335, E3 +52577.995}
SPL {X  -139.539, Y  +757.399, Z    +0.000, E1   -73.892, E3 +52584.192}
SPL {X  -136.017, Y  +762.997, Z    +0.000, E1   -73.579, E3 +52589.375}
SPL {X  -133.089, Y  +767.296, Z    +0.000, E1   -73.251, E3 +52593.833}
SPL {X  -129.985, Y  +771.553, Z    +0.000, E1   -72.801, E3 +52598.827}
SPL {X  -126.581, Y  +775.909, Z    +0.000, E1   -72.426, E3 +52603.138}
SPL {X  -123.329, Y  +779.803, Z    +0.000, E1   -71.936, E3 +52607.520}
SPL {X  -119.291, Y  +784.315, Z    +0.000, E1   -72.148, E3 +52608.932}
SPL {X   -57.587, Y  +825.796, Z    +0.000, E1   -56.753, E3 +52762.694}
ENDSPLINE

